   me.stations[22].raw[43,4] := WSTRING#'';
   me.stations[22].raw[43,5] := WSTRING#'';
   me.stations[22].raw[43,6] := WSTRING#'';
   me.stations[22].raw[43,7] := WSTRING#'';
   me.stations[22].raw[44,0] := WSTRING#'';
   me.stations[22].raw[44,1] := WSTRING#'';
   me.stations[22].raw[44,2] := WSTRING#'';
   me.stations[22].raw[44,3] := WSTRING#'';
   me.stations[22].raw[44,4] := WSTRING#'';
   me.stations[22].raw[44,5] := WSTRING#'';
   me.stations[22].raw[44,6] := WSTRING#'';
   me.stations[22].raw[44,7] := WSTRING#'';
   me.stations[22].raw[45,0] := WSTRING#'';
   me.stations[22].raw[45,1] := WSTRING#'';
   me.stations[22].raw[45,2] := WSTRING#'';
   me.stations[22].raw[45,3] := WSTRING#'';
   me.stations[22].raw[45,4] := WSTRING#'';
   me.stations[22].raw[45,5] := WSTRING#'';
   me.stations[22].raw[45,6] := WSTRING#'';
   me.stations[22].raw[45,7] := WSTRING#'';
   me.stations[22].raw[46,0] := WSTRING#'';
   me.stations[22].raw[46,1] := WSTRING#'';
   me.stations[22].raw[46,2] := WSTRING#'';
   me.stations[22].raw[46,3] := WSTRING#'';
   me.stations[22].raw[46,4] := WSTRING#'';
   me.stations[22].raw[46,5] := WSTRING#'';
   me.stations[22].raw[46,6] := WSTRING#'';
   me.stations[22].raw[46,7] := WSTRING#'';
   me.stations[22].raw[47,0] := WSTRING#'';
   me.stations[22].raw[47,1] := WSTRING#'';
   me.stations[22].raw[47,2] := WSTRING#'';
   me.stations[22].raw[47,3] := WSTRING#'';
   me.stations[22].raw[47,4] := WSTRING#'';
   me.stations[22].raw[47,5] := WSTRING#'';
   me.stations[22].raw[47,6] := WSTRING#'';
   me.stations[22].raw[47,7] := WSTRING#'';
   me.stations[22].raw[48,0] := WSTRING#'';
   me.stations[22].raw[48,1] := WSTRING#'';
   me.stations[22].raw[48,2] := WSTRING#'';
   me.stations[22].raw[48,3] := WSTRING#'';
   me.stations[22].raw[48,4] := WSTRING#'';
   me.stations[22].raw[48,5] := WSTRING#'';
   me.stations[22].raw[48,6] := WSTRING#'';
   me.stations[22].raw[48,7] := WSTRING#'';
   me.stations[22].raw[49,0] := WSTRING#'';
   me.stations[22].raw[49,1] := WSTRING#'';
   me.stations[22].raw[49,2] := WSTRING#'';
   me.stations[22].raw[49,3] := WSTRING#'';
   me.stations[22].raw[49,4] := WSTRING#'';
   me.stations[22].raw[49,5] := WSTRING#'';
   me.stations[22].raw[49,6] := WSTRING#'';
   me.stations[22].raw[49,7] := WSTRING#'';
   me.stations[23].size := 0;
   me.stations[23].wip[0] := WSTRING#'';
   me.stations[23].wip[1] := WSTRING#'';
   me.stations[23].wip[2] := WSTRING#'';
   me.stations[23].wip[3] := WSTRING#'';
   me.stations[23].wip[4] := WSTRING#'';
   me.stations[23].wip[5] := WSTRING#'';
   me.stations[23].wip[6] := WSTRING#'';
   me.stations[23].wip[7] := WSTRING#'';
   me.stations[23].wip[8] := WSTRING#'';
   me.stations[23].wip[9] := WSTRING#'';
   me.stations[23].wip[10] := WSTRING#'';
   me.stations[23].wip[11] := WSTRING#'';
   me.stations[23].wip[12] := WSTRING#'';
   me.stations[23].wip[13] := WSTRING#'';
   me.stations[23].wip[14] := WSTRING#'';
   me.stations[23].wip[15] := WSTRING#'';
   me.stations[23].wip[16] := WSTRING#'';
   me.stations[23].wip[17] := WSTRING#'';
   me.stations[23].wip[18] := WSTRING#'';
   me.stations[23].wip[19] := WSTRING#'';
   me.stations[23].wip[20] := WSTRING#'';
   me.stations[23].wip[21] := WSTRING#'';
   me.stations[23].wip[22] := WSTRING#'';
   me.stations[23].wip[23] := WSTRING#'';
   me.stations[23].wip[24] := WSTRING#'';
   me.stations[23].wip[25] := WSTRING#'';
   me.stations[23].wip[26] := WSTRING#'';
   me.stations[23].wip[27] := WSTRING#'';
   me.stations[23].wip[28] := WSTRING#'';
   me.stations[23].wip[29] := WSTRING#'';
   me.stations[23].wip[30] := WSTRING#'';
   me.stations[23].wip[31] := WSTRING#'';
   me.stations[23].wip[32] := WSTRING#'';
   me.stations[23].wip[33] := WSTRING#'';
   me.stations[23].wip[34] := WSTRING#'';
   me.stations[23].wip[35] := WSTRING#'';
   me.stations[23].wip[36] := WSTRING#'';
   me.stations[23].wip[37] := WSTRING#'';
   me.stations[23].wip[38] := WSTRING#'';
   me.stations[23].wip[39] := WSTRING#'';
   me.stations[23].wip[40] := WSTRING#'';
   me.stations[23].wip[41] := WSTRING#'';
   me.stations[23].wip[42] := WSTRING#'';
   me.stations[23].wip[43] := WSTRING#'';
   me.stations[23].wip[44] := WSTRING#'';
   me.stations[23].wip[45] := WSTRING#'';
   me.stations[23].wip[46] := WSTRING#'';
   me.stations[23].wip[47] := WSTRING#'';
   me.stations[23].wip[48] := WSTRING#'';
   me.stations[23].wip[49] := WSTRING#'';
   me.stations[23].raw[0,0] := WSTRING#'';
   me.stations[23].raw[0,1] := WSTRING#'';
   me.stations[23].raw[0,2] := WSTRING#'';
   me.stations[23].raw[0,3] := WSTRING#'';
   me.stations[23].raw[0,4] := WSTRING#'';
   me.stations[23].raw[0,5] := WSTRING#'';
   me.stations[23].raw[0,6] := WSTRING#'';
   me.stations[23].raw[0,7] := WSTRING#'';
   me.stations[23].raw[1,0] := WSTRING#'';
   me.stations[23].raw[1,1] := WSTRING#'';
   me.stations[23].raw[1,2] := WSTRING#'';
   me.stations[23].raw[1,3] := WSTRING#'';
   me.stations[23].raw[1,4] := WSTRING#'';
   me.stations[23].raw[1,5] := WSTRING#'';
   me.stations[23].raw[1,6] := WSTRING#'';
   me.stations[23].raw[1,7] := WSTRING#'';
   me.stations[23].raw[2,0] := WSTRING#'';
   me.stations[23].raw[2,1] := WSTRING#'';
   me.stations[23].raw[2,2] := WSTRING#'';
   me.stations[23].raw[2,3] := WSTRING#'';
   me.stations[23].raw[2,4] := WSTRING#'';
   me.stations[23].raw[2,5] := WSTRING#'';
   me.stations[23].raw[2,6] := WSTRING#'';
   me.stations[23].raw[2,7] := WSTRING#'';
   me.stations[23].raw[3,0] := WSTRING#'';
   me.stations[23].raw[3,1] := WSTRING#'';
   me.stations[23].raw[3,2] := WSTRING#'';
   me.stations[23].raw[3,3] := WSTRING#'';
   me.stations[23].raw[3,4] := WSTRING#'';
   me.stations[23].raw[3,5] := WSTRING#'';
   me.stations[23].raw[3,6] := WSTRING#'';
   me.stations[23].raw[3,7] := WSTRING#'';
   me.stations[23].raw[4,0] := WSTRING#'';
   me.stations[23].raw[4,1] := WSTRING#'';
   me.stations[23].raw[4,2] := WSTRING#'';
   me.stations[23].raw[4,3] := WSTRING#'';
   me.stations[23].raw[4,4] := WSTRING#'';
   me.stations[23].raw[4,5] := WSTRING#'';
   me.stations[23].raw[4,6] := WSTRING#'';
   me.stations[23].raw[4,7] := WSTRING#'';
   me.stations[23].raw[5,0] := WSTRING#'';
   me.stations[23].raw[5,1] := WSTRING#'';
   me.stations[23].raw[5,2] := WSTRING#'';
   me.stations[23].raw[5,3] := WSTRING#'';
   me.stations[23].raw[5,4] := WSTRING#'';
   me.stations[23].raw[5,5] := WSTRING#'';
   me.stations[23].raw[5,6] := WSTRING#'';
   me.stations[23].raw[5,7] := WSTRING#'';
   me.stations[23].raw[6,0] := WSTRING#'';
   me.stations[23].raw[6,1] := WSTRING#'';
   me.stations[23].raw[6,2] := WSTRING#'';
   me.stations[23].raw[6,3] := WSTRING#'';
   me.stations[23].raw[6,4] := WSTRING#'';
   me.stations[23].raw[6,5] := WSTRING#'';
   me.stations[23].raw[6,6] := WSTRING#'';
   me.stations[23].raw[6,7] := WSTRING#'';
   me.stations[23].raw[7,0] := WSTRING#'';
   me.stations[23].raw[7,1] := WSTRING#'';
   me.stations[23].raw[7,2] := WSTRING#'';
   me.stations[23].raw[7,3] := WSTRING#'';
   me.stations[23].raw[7,4] := WSTRING#'';
   me.stations[23].raw[7,5] := WSTRING#'';
   me.stations[23].raw[7,6] := WSTRING#'';
   me.stations[23].raw[7,7] := WSTRING#'';
   me.stations[23].raw[8,0] := WSTRING#'';
   me.stations[23].raw[8,1] := WSTRING#'';
   me.stations[23].raw[8,2] := WSTRING#'';
   me.stations[23].raw[8,3] := WSTRING#'';
   me.stations[23].raw[8,4] := WSTRING#'';
   me.stations[23].raw[8,5] := WSTRING#'';
   me.stations[23].raw[8,6] := WSTRING#'';
   me.stations[23].raw[8,7] := WSTRING#'';
   me.stations[23].raw[9,0] := WSTRING#'';
   me.stations[23].raw[9,1] := WSTRING#'';
   me.stations[23].raw[9,2] := WSTRING#'';
   me.stations[23].raw[9,3] := WSTRING#'';
   me.stations[23].raw[9,4] := WSTRING#'';
   me.stations[23].raw[9,5] := WSTRING#'';
   me.stations[23].raw[9,6] := WSTRING#'';
   me.stations[23].raw[9,7] := WSTRING#'';
   me.stations[23].raw[10,0] := WSTRING#'';
   me.stations[23].raw[10,1] := WSTRING#'';
   me.stations[23].raw[10,2] := WSTRING#'';
   me.stations[23].raw[10,3] := WSTRING#'';
   me.stations[23].raw[10,4] := WSTRING#'';
   me.stations[23].raw[10,5] := WSTRING#'';
   me.stations[23].raw[10,6] := WSTRING#'';
   me.stations[23].raw[10,7] := WSTRING#'';
   me.stations[23].raw[11,0] := WSTRING#'';
   me.stations[23].raw[11,1] := WSTRING#'';
   me.stations[23].raw[11,2] := WSTRING#'';
   me.stations[23].raw[11,3] := WSTRING#'';
   me.stations[23].raw[11,4] := WSTRING#'';
   me.stations[23].raw[11,5] := WSTRING#'';
   me.stations[23].raw[11,6] := WSTRING#'';
   me.stations[23].raw[11,7] := WSTRING#'';
   me.stations[23].raw[12,0] := WSTRING#'';
   me.stations[23].raw[12,1] := WSTRING#'';
   me.stations[23].raw[12,2] := WSTRING#'';
   me.stations[23].raw[12,3] := WSTRING#'';
   me.stations[23].raw[12,4] := WSTRING#'';
   me.stations[23].raw[12,5] := WSTRING#'';
   me.stations[23].raw[12,6] := WSTRING#'';
   me.stations[23].raw[12,7] := WSTRING#'';
   me.stations[23].raw[13,0] := WSTRING#'';
   me.stations[23].raw[13,1] := WSTRING#'';
   me.stations[23].raw[13,2] := WSTRING#'';
   me.stations[23].raw[13,3] := WSTRING#'';
   me.stations[23].raw[13,4] := WSTRING#'';
   me.stations[23].raw[13,5] := WSTRING#'';
   me.stations[23].raw[13,6] := WSTRING#'';
   me.stations[23].raw[13,7] := WSTRING#'';
   me.stations[23].raw[14,0] := WSTRING#'';
   me.stations[23].raw[14,1] := WSTRING#'';
   me.stations[23].raw[14,2] := WSTRING#'';
   me.stations[23].raw[14,3] := WSTRING#'';
   me.stations[23].raw[14,4] := WSTRING#'';
   me.stations[23].raw[14,5] := WSTRING#'';
   me.stations[23].raw[14,6] := WSTRING#'';
   me.stations[23].raw[14,7] := WSTRING#'';
   me.stations[23].raw[15,0] := WSTRING#'';
   me.stations[23].raw[15,1] := WSTRING#'';
   me.stations[23].raw[15,2] := WSTRING#'';
   me.stations[23].raw[15,3] := WSTRING#'';
   me.stations[23].raw[15,4] := WSTRING#'';
   me.stations[23].raw[15,5] := WSTRING#'';
   me.stations[23].raw[15,6] := WSTRING#'';
   me.stations[23].raw[15,7] := WSTRING#'';
   me.stations[23].raw[16,0] := WSTRING#'';
   me.stations[23].raw[16,1] := WSTRING#'';
   me.stations[23].raw[16,2] := WSTRING#'';
   me.stations[23].raw[16,3] := WSTRING#'';
   me.stations[23].raw[16,4] := WSTRING#'';
   me.stations[23].raw[16,5] := WSTRING#'';
   me.stations[23].raw[16,6] := WSTRING#'';
   me.stations[23].raw[16,7] := WSTRING#'';
   me.stations[23].raw[17,0] := WSTRING#'';
   me.stations[23].raw[17,1] := WSTRING#'';
   me.stations[23].raw[17,2] := WSTRING#'';
   me.stations[23].raw[17,3] := WSTRING#'';
   me.stations[23].raw[17,4] := WSTRING#'';
   me.stations[23].raw[17,5] := WSTRING#'';
   me.stations[23].raw[17,6] := WSTRING#'';
   me.stations[23].raw[17,7] := WSTRING#'';
   me.stations[23].raw[18,0] := WSTRING#'';
   me.stations[23].raw[18,1] := WSTRING#'';
   me.stations[23].raw[18,2] := WSTRING#'';
   me.stations[23].raw[18,3] := WSTRING#'';
   me.stations[23].raw[18,4] := WSTRING#'';
   me.stations[23].raw[18,5] := WSTRING#'';
   me.stations[23].raw[18,6] := WSTRING#'';
   me.stations[23].raw[18,7] := WSTRING#'';
   me.stations[23].raw[19,0] := WSTRING#'';
   me.stations[23].raw[19,1] := WSTRING#'';
   me.stations[23].raw[19,2] := WSTRING#'';
   me.stations[23].raw[19,3] := WSTRING#'';
   me.stations[23].raw[19,4] := WSTRING#'';
   me.stations[23].raw[19,5] := WSTRING#'';
   me.stations[23].raw[19,6] := WSTRING#'';
   me.stations[23].raw[19,7] := WSTRING#'';
   me.stations[23].raw[20,0] := WSTRING#'';
   me.stations[23].raw[20,1] := WSTRING#'';
   me.stations[23].raw[20,2] := WSTRING#'';
   me.stations[23].raw[20,3] := WSTRING#'';
   me.stations[23].raw[20,4] := WSTRING#'';
   me.stations[23].raw[20,5] := WSTRING#'';
   me.stations[23].raw[20,6] := WSTRING#'';
   me.stations[23].raw[20,7] := WSTRING#'';
   me.stations[23].raw[21,0] := WSTRING#'';
   me.stations[23].raw[21,1] := WSTRING#'';
   me.stations[23].raw[21,2] := WSTRING#'';
   me.stations[23].raw[21,3] := WSTRING#'';
   me.stations[23].raw[21,4] := WSTRING#'';
   me.stations[23].raw[21,5] := WSTRING#'';
   me.stations[23].raw[21,6] := WSTRING#'';
   me.stations[23].raw[21,7] := WSTRING#'';
   me.stations[23].raw[22,0] := WSTRING#'';
   me.stations[23].raw[22,1] := WSTRING#'';
   me.stations[23].raw[22,2] := WSTRING#'';
   me.stations[23].raw[22,3] := WSTRING#'';
   me.stations[23].raw[22,4] := WSTRING#'';
   me.stations[23].raw[22,5] := WSTRING#'';
   me.stations[23].raw[22,6] := WSTRING#'';
   me.stations[23].raw[22,7] := WSTRING#'';
   me.stations[23].raw[23,0] := WSTRING#'';
   me.stations[23].raw[23,1] := WSTRING#'';
   me.stations[23].raw[23,2] := WSTRING#'';
   me.stations[23].raw[23,3] := WSTRING#'';
   me.stations[23].raw[23,4] := WSTRING#'';
   me.stations[23].raw[23,5] := WSTRING#'';
   me.stations[23].raw[23,6] := WSTRING#'';
   me.stations[23].raw[23,7] := WSTRING#'';
   me.stations[23].raw[24,0] := WSTRING#'';
   me.stations[23].raw[24,1] := WSTRING#'';
   me.stations[23].raw[24,2] := WSTRING#'';
   me.stations[23].raw[24,3] := WSTRING#'';
   me.stations[23].raw[24,4] := WSTRING#'';
   me.stations[23].raw[24,5] := WSTRING#'';
   me.stations[23].raw[24,6] := WSTRING#'';
   me.stations[23].raw[24,7] := WSTRING#'';
   me.stations[23].raw[25,0] := WSTRING#'';
   me.stations[23].raw[25,1] := WSTRING#'';
   me.stations[23].raw[25,2] := WSTRING#'';
   me.stations[23].raw[25,3] := WSTRING#'';
   me.stations[23].raw[25,4] := WSTRING#'';
   me.stations[23].raw[25,5] := WSTRING#'';
   me.stations[23].raw[25,6] := WSTRING#'';
   me.stations[23].raw[25,7] := WSTRING#'';
   me.stations[23].raw[26,0] := WSTRING#'';
   me.stations[23].raw[26,1] := WSTRING#'';
   me.stations[23].raw[26,2] := WSTRING#'';
   me.stations[23].raw[26,3] := WSTRING#'';
   me.stations[23].raw[26,4] := WSTRING#'';
   me.stations[23].raw[26,5] := WSTRING#'';
   me.stations[23].raw[26,6] := WSTRING#'';
   me.stations[23].raw[26,7] := WSTRING#'';
   me.stations[23].raw[27,0] := WSTRING#'';
   me.stations[23].raw[27,1] := WSTRING#'';
   me.stations[23].raw[27,2] := WSTRING#'';
   me.stations[23].raw[27,3] := WSTRING#'';
   me.stations[23].raw[27,4] := WSTRING#'';
   me.stations[23].raw[27,5] := WSTRING#'';
   me.stations[23].raw[27,6] := WSTRING#'';
   me.stations[23].raw[27,7] := WSTRING#'';
   me.stations[23].raw[28,0] := WSTRING#'';
   me.stations[23].raw[28,1] := WSTRING#'';
   me.stations[23].raw[28,2] := WSTRING#'';
   me.stations[23].raw[28,3] := WSTRING#'';
   me.stations[23].raw[28,4] := WSTRING#'';
   me.stations[23].raw[28,5] := WSTRING#'';
   me.stations[23].raw[28,6] := WSTRING#'';
   me.stations[23].raw[28,7] := WSTRING#'';
   me.stations[23].raw[29,0] := WSTRING#'';
   me.stations[23].raw[29,1] := WSTRING#'';
   me.stations[23].raw[29,2] := WSTRING#'';
   me.stations[23].raw[29,3] := WSTRING#'';
   me.stations[23].raw[29,4] := WSTRING#'';
   me.stations[23].raw[29,5] := WSTRING#'';
   me.stations[23].raw[29,6] := WSTRING#'';
   me.stations[23].raw[29,7] := WSTRING#'';
   me.stations[23].raw[30,0] := WSTRING#'';
   me.stations[23].raw[30,1] := WSTRING#'';
   me.stations[23].raw[30,2] := WSTRING#'';
   me.stations[23].raw[30,3] := WSTRING#'';
   me.stations[23].raw[30,4] := WSTRING#'';
   me.stations[23].raw[30,5] := WSTRING#'';
   me.stations[23].raw[30,6] := WSTRING#'';
   me.stations[23].raw[30,7] := WSTRING#'';
   me.stations[23].raw[31,0] := WSTRING#'';
   me.stations[23].raw[31,1] := WSTRING#'';
   me.stations[23].raw[31,2] := WSTRING#'';
   me.stations[23].raw[31,3] := WSTRING#'';
   me.stations[23].raw[31,4] := WSTRING#'';
   me.stations[23].raw[31,5] := WSTRING#'';
   me.stations[23].raw[31,6] := WSTRING#'';
   me.stations[23].raw[31,7] := WSTRING#'';
   me.stations[23].raw[32,0] := WSTRING#'';
   me.stations[23].raw[32,1] := WSTRING#'';
   me.stations[23].raw[32,2] := WSTRING#'';
   me.stations[23].raw[32,3] := WSTRING#'';
   me.stations[23].raw[32,4] := WSTRING#'';
   me.stations[23].raw[32,5] := WSTRING#'';
   me.stations[23].raw[32,6] := WSTRING#'';
   me.stations[23].raw[32,7] := WSTRING#'';
   me.stations[23].raw[33,0] := WSTRING#'';
   me.stations[23].raw[33,1] := WSTRING#'';
   me.stations[23].raw[33,2] := WSTRING#'';
   me.stations[23].raw[33,3] := WSTRING#'';
   me.stations[23].raw[33,4] := WSTRING#'';
   me.stations[23].raw[33,5] := WSTRING#'';
   me.stations[23].raw[33,6] := WSTRING#'';
   me.stations[23].raw[33,7] := WSTRING#'';
   me.stations[23].raw[34,0] := WSTRING#'';
   me.stations[23].raw[34,1] := WSTRING#'';
   me.stations[23].raw[34,2] := WSTRING#'';
   me.stations[23].raw[34,3] := WSTRING#'';
   me.stations[23].raw[34,4] := WSTRING#'';
   me.stations[23].raw[34,5] := WSTRING#'';
   me.stations[23].raw[34,6] := WSTRING#'';
   me.stations[23].raw[34,7] := WSTRING#'';
   me.stations[23].raw[35,0] := WSTRING#'';
   me.stations[23].raw[35,1] := WSTRING#'';
   me.stations[23].raw[35,2] := WSTRING#'';
   me.stations[23].raw[35,3] := WSTRING#'';
   me.stations[23].raw[35,4] := WSTRING#'';
   me.stations[23].raw[35,5] := WSTRING#'';
   me.stations[23].raw[35,6] := WSTRING#'';
   me.stations[23].raw[35,7] := WSTRING#'';
   me.stations[23].raw[36,0] := WSTRING#'';
   me.stations[23].raw[36,1] := WSTRING#'';
   me.stations[23].raw[36,2] := WSTRING#'';
   me.stations[23].raw[36,3] := WSTRING#'';
   me.stations[23].raw[36,4] := WSTRING#'';
   me.stations[23].raw[36,5] := WSTRING#'';
   me.stations[23].raw[36,6] := WSTRING#'';
   me.stations[23].raw[36,7] := WSTRING#'';
   me.stations[23].raw[37,0] := WSTRING#'';
   me.stations[23].raw[37,1] := WSTRING#'';
   me.stations[23].raw[37,2] := WSTRING#'';
   me.stations[23].raw[37,3] := WSTRING#'';
   me.stations[23].raw[37,4] := WSTRING#'';
   me.stations[23].raw[37,5] := WSTRING#'';
   me.stations[23].raw[37,6] := WSTRING#'';
   me.stations[23].raw[37,7] := WSTRING#'';
   me.stations[23].raw[38,0] := WSTRING#'';
   me.stations[23].raw[38,1] := WSTRING#'';
   me.stations[23].raw[38,2] := WSTRING#'';
   me.stations[23].raw[38,3] := WSTRING#'';
   me.stations[23].raw[38,4] := WSTRING#'';
   me.stations[23].raw[38,5] := WSTRING#'';
   me.stations[23].raw[38,6] := WSTRING#'';
   me.stations[23].raw[38,7] := WSTRING#'';
   me.stations[23].raw[39,0] := WSTRING#'';
   me.stations[23].raw[39,1] := WSTRING#'';
   me.stations[23].raw[39,2] := WSTRING#'';
   me.stations[23].raw[39,3] := WSTRING#'';
   me.stations[23].raw[39,4] := WSTRING#'';
   me.stations[23].raw[39,5] := WSTRING#'';
   me.stations[23].raw[39,6] := WSTRING#'';
   me.stations[23].raw[39,7] := WSTRING#'';
   me.stations[23].raw[40,0] := WSTRING#'';
   me.stations[23].raw[40,1] := WSTRING#'';
   me.stations[23].raw[40,2] := WSTRING#'';
   me.stations[23].raw[40,3] := WSTRING#'';
   me.stations[23].raw[40,4] := WSTRING#'';
   me.stations[23].raw[40,5] := WSTRING#'';
   me.stations[23].raw[40,6] := WSTRING#'';
   me.stations[23].raw[40,7] := WSTRING#'';
   me.stations[23].raw[41,0] := WSTRING#'';
   me.stations[23].raw[41,1] := WSTRING#'';
   me.stations[23].raw[41,2] := WSTRING#'';
   me.stations[23].raw[41,3] := WSTRING#'';
   me.stations[23].raw[41,4] := WSTRING#'';
   me.stations[23].raw[41,5] := WSTRING#'';
   me.stations[23].raw[41,6] := WSTRING#'';
   me.stations[23].raw[41,7] := WSTRING#'';
   me.stations[23].raw[42,0] := WSTRING#'';
   me.stations[23].raw[42,1] := WSTRING#'';
   me.stations[23].raw[42,2] := WSTRING#'';
   me.stations[23].raw[42,3] := WSTRING#'';
   me.stations[23].raw[42,4] := WSTRING#'';
   me.stations[23].raw[42,5] := WSTRING#'';
   me.stations[23].raw[42,6] := WSTRING#'';
   me.stations[23].raw[42,7] := WSTRING#'';
   me.stations[23].raw[43,0] := WSTRING#'';
   me.stations[23].raw[43,1] := WSTRING#'';
   me.stations[23].raw[43,2] := WSTRING#'';
   me.stations[23].raw[43,3] := WSTRING#'';
   me.stations[23].raw[43,4] := WSTRING#'';
   me.stations[23].raw[43,5] := WSTRING#'';
   me.stations[23].raw[43,6] := WSTRING#'';
   me.stations[23].raw[43,7] := WSTRING#'';
   me.stations[23].raw[44,0] := WSTRING#'';
   me.stations[23].raw[44,1] := WSTRING#'';
   me.stations[23].raw[44,2] := WSTRING#'';
   me.stations[23].raw[44,3] := WSTRING#'';
   me.stations[23].raw[44,4] := WSTRING#'';
   me.stations[23].raw[44,5] := WSTRING#'';
   me.stations[23].raw[44,6] := WSTRING#'';
   me.stations[23].raw[44,7] := WSTRING#'';
   me.stations[23].raw[45,0] := WSTRING#'';
   me.stations[23].raw[45,1] := WSTRING#'';
   me.stations[23].raw[45,2] := WSTRING#'';
   me.stations[23].raw[45,3] := WSTRING#'';
   me.stations[23].raw[45,4] := WSTRING#'';
   me.stations[23].raw[45,5] := WSTRING#'';
   me.stations[23].raw[45,6] := WSTRING#'';
   me.stations[23].raw[45,7] := WSTRING#'';
   me.stations[23].raw[46,0] := WSTRING#'';
   me.stations[23].raw[46,1] := WSTRING#'';
   me.stations[23].raw[46,2] := WSTRING#'';
   me.stations[23].raw[46,3] := WSTRING#'';
   me.stations[23].raw[46,4] := WSTRING#'';
   me.stations[23].raw[46,5] := WSTRING#'';
   me.stations[23].raw[46,6] := WSTRING#'';
   me.stations[23].raw[46,7] := WSTRING#'';
   me.stations[23].raw[47,0] := WSTRING#'';
   me.stations[23].raw[47,1] := WSTRING#'';
   me.stations[23].raw[47,2] := WSTRING#'';
   me.stations[23].raw[47,3] := WSTRING#'';
   me.stations[23].raw[47,4] := WSTRING#'';
   me.stations[23].raw[47,5] := WSTRING#'';
   me.stations[23].raw[47,6] := WSTRING#'';
   me.stations[23].raw[47,7] := WSTRING#'';
   me.stations[23].raw[48,0] := WSTRING#'';
   me.stations[23].raw[48,1] := WSTRING#'';
   me.stations[23].raw[48,2] := WSTRING#'';
   me.stations[23].raw[48,3] := WSTRING#'';
   me.stations[23].raw[48,4] := WSTRING#'';
   me.stations[23].raw[48,5] := WSTRING#'';
   me.stations[23].raw[48,6] := WSTRING#'';
   me.stations[23].raw[48,7] := WSTRING#'';
   me.stations[23].raw[49,0] := WSTRING#'';
   me.stations[23].raw[49,1] := WSTRING#'';
   me.stations[23].raw[49,2] := WSTRING#'';
   me.stations[23].raw[49,3] := WSTRING#'';
   me.stations[23].raw[49,4] := WSTRING#'';
   me.stations[23].raw[49,5] := WSTRING#'';
   me.stations[23].raw[49,6] := WSTRING#'';
   me.stations[23].raw[49,7] := WSTRING#'';
   me.stations[24].size := 0;
   me.stations[24].wip[0] := WSTRING#'';
   me.stations[24].wip[1] := WSTRING#'';
   me.stations[24].wip[2] := WSTRING#'';
   me.stations[24].wip[3] := WSTRING#'';
   me.stations[24].wip[4] := WSTRING#'';
   me.stations[24].wip[5] := WSTRING#'';
   me.stations[24].wip[6] := WSTRING#'';
   me.stations[24].wip[7] := WSTRING#'';
   me.stations[24].wip[8] := WSTRING#'';
   me.stations[24].wip[9] := WSTRING#'';
   me.stations[24].wip[10] := WSTRING#'';
   me.stations[24].wip[11] := WSTRING#'';
   me.stations[24].wip[12] := WSTRING#'';
   me.stations[24].wip[13] := WSTRING#'';
   me.stations[24].wip[14] := WSTRING#'';
   me.stations[24].wip[15] := WSTRING#'';
   me.stations[24].wip[16] := WSTRING#'';
   me.stations[24].wip[17] := WSTRING#'';
   me.stations[24].wip[18] := WSTRING#'';
   me.stations[24].wip[19] := WSTRING#'';
   me.stations[24].wip[20] := WSTRING#'';
   me.stations[24].wip[21] := WSTRING#'';
   me.stations[24].wip[22] := WSTRING#'';
   me.stations[24].wip[23] := WSTRING#'';
   me.stations[24].wip[24] := WSTRING#'';
   me.stations[24].wip[25] := WSTRING#'';
   me.stations[24].wip[26] := WSTRING#'';
   me.stations[24].wip[27] := WSTRING#'';
   me.stations[24].wip[28] := WSTRING#'';
   me.stations[24].wip[29] := WSTRING#'';
   me.stations[24].wip[30] := WSTRING#'';
   me.stations[24].wip[31] := WSTRING#'';
   me.stations[24].wip[32] := WSTRING#'';
   me.stations[24].wip[33] := WSTRING#'';
   me.stations[24].wip[34] := WSTRING#'';
   me.stations[24].wip[35] := WSTRING#'';
   me.stations[24].wip[36] := WSTRING#'';
   me.stations[24].wip[37] := WSTRING#'';
   me.stations[24].wip[38] := WSTRING#'';
   me.stations[24].wip[39] := WSTRING#'';
   me.stations[24].wip[40] := WSTRING#'';
   me.stations[24].wip[41] := WSTRING#'';
   me.stations[24].wip[42] := WSTRING#'';
   me.stations[24].wip[43] := WSTRING#'';
   me.stations[24].wip[44] := WSTRING#'';
   me.stations[24].wip[45] := WSTRING#'';
   me.stations[24].wip[46] := WSTRING#'';
   me.stations[24].wip[47] := WSTRING#'';
   me.stations[24].wip[48] := WSTRING#'';
   me.stations[24].wip[49] := WSTRING#'';
   me.stations[24].raw[0,0] := WSTRING#'';
   me.stations[24].raw[0,1] := WSTRING#'';
   me.stations[24].raw[0,2] := WSTRING#'';
   me.stations[24].raw[0,3] := WSTRING#'';
   me.stations[24].raw[0,4] := WSTRING#'';
   me.stations[24].raw[0,5] := WSTRING#'';
   me.stations[24].raw[0,6] := WSTRING#'';
   me.stations[24].raw[0,7] := WSTRING#'';
   me.stations[24].raw[1,0] := WSTRING#'';
   me.stations[24].raw[1,1] := WSTRING#'';
   me.stations[24].raw[1,2] := WSTRING#'';
   me.stations[24].raw[1,3] := WSTRING#'';
   me.stations[24].raw[1,4] := WSTRING#'';
   me.stations[24].raw[1,5] := WSTRING#'';
   me.stations[24].raw[1,6] := WSTRING#'';
   me.stations[24].raw[1,7] := WSTRING#'';
   me.stations[24].raw[2,0] := WSTRING#'';
   me.stations[24].raw[2,1] := WSTRING#'';
   me.stations[24].raw[2,2] := WSTRING#'';
   me.stations[24].raw[2,3] := WSTRING#'';
   me.stations[24].raw[2,4] := WSTRING#'';
   me.stations[24].raw[2,5] := WSTRING#'';
   me.stations[24].raw[2,6] := WSTRING#'';
   me.stations[24].raw[2,7] := WSTRING#'';
   me.stations[24].raw[3,0] := WSTRING#'';
   me.stations[24].raw[3,1] := WSTRING#'';
   me.stations[24].raw[3,2] := WSTRING#'';
   me.stations[24].raw[3,3] := WSTRING#'';
   me.stations[24].raw[3,4] := WSTRING#'';
   me.stations[24].raw[3,5] := WSTRING#'';
   me.stations[24].raw[3,6] := WSTRING#'';
   me.stations[24].raw[3,7] := WSTRING#'';
   me.stations[24].raw[4,0] := WSTRING#'';
   me.stations[24].raw[4,1] := WSTRING#'';
   me.stations[24].raw[4,2] := WSTRING#'';
   me.stations[24].raw[4,3] := WSTRING#'';
   me.stations[24].raw[4,4] := WSTRING#'';
   me.stations[24].raw[4,5] := WSTRING#'';
   me.stations[24].raw[4,6] := WSTRING#'';
   me.stations[24].raw[4,7] := WSTRING#'';
   me.stations[24].raw[5,0] := WSTRING#'';
   me.stations[24].raw[5,1] := WSTRING#'';
   me.stations[24].raw[5,2] := WSTRING#'';
   me.stations[24].raw[5,3] := WSTRING#'';
   me.stations[24].raw[5,4] := WSTRING#'';
   me.stations[24].raw[5,5] := WSTRING#'';
   me.stations[24].raw[5,6] := WSTRING#'';
   me.stations[24].raw[5,7] := WSTRING#'';
   me.stations[24].raw[6,0] := WSTRING#'';
   me.stations[24].raw[6,1] := WSTRING#'';
   me.stations[24].raw[6,2] := WSTRING#'';
   me.stations[24].raw[6,3] := WSTRING#'';
   me.stations[24].raw[6,4] := WSTRING#'';
   me.stations[24].raw[6,5] := WSTRING#'';
   me.stations[24].raw[6,6] := WSTRING#'';
   me.stations[24].raw[6,7] := WSTRING#'';
   me.stations[24].raw[7,0] := WSTRING#'';
   me.stations[24].raw[7,1] := WSTRING#'';
   me.stations[24].raw[7,2] := WSTRING#'';
   me.stations[24].raw[7,3] := WSTRING#'';
   me.stations[24].raw[7,4] := WSTRING#'';
   me.stations[24].raw[7,5] := WSTRING#'';
   me.stations[24].raw[7,6] := WSTRING#'';
   me.stations[24].raw[7,7] := WSTRING#'';
   me.stations[24].raw[8,0] := WSTRING#'';
   me.stations[24].raw[8,1] := WSTRING#'';
   me.stations[24].raw[8,2] := WSTRING#'';
   me.stations[24].raw[8,3] := WSTRING#'';
   me.stations[24].raw[8,4] := WSTRING#'';
   me.stations[24].raw[8,5] := WSTRING#'';
   me.stations[24].raw[8,6] := WSTRING#'';
   me.stations[24].raw[8,7] := WSTRING#'';
   me.stations[24].raw[9,0] := WSTRING#'';
   me.stations[24].raw[9,1] := WSTRING#'';
   me.stations[24].raw[9,2] := WSTRING#'';
   me.stations[24].raw[9,3] := WSTRING#'';
   me.stations[24].raw[9,4] := WSTRING#'';
   me.stations[24].raw[9,5] := WSTRING#'';
   me.stations[24].raw[9,6] := WSTRING#'';
   me.stations[24].raw[9,7] := WSTRING#'';
   me.stations[24].raw[10,0] := WSTRING#'';
   me.stations[24].raw[10,1] := WSTRING#'';
   me.stations[24].raw[10,2] := WSTRING#'';
   me.stations[24].raw[10,3] := WSTRING#'';
   me.stations[24].raw[10,4] := WSTRING#'';
   me.stations[24].raw[10,5] := WSTRING#'';
   me.stations[24].raw[10,6] := WSTRING#'';
   me.stations[24].raw[10,7] := WSTRING#'';
   me.stations[24].raw[11,0] := WSTRING#'';
   me.stations[24].raw[11,1] := WSTRING#'';
   me.stations[24].raw[11,2] := WSTRING#'';
   me.stations[24].raw[11,3] := WSTRING#'';
   me.stations[24].raw[11,4] := WSTRING#'';
   me.stations[24].raw[11,5] := WSTRING#'';
   me.stations[24].raw[11,6] := WSTRING#'';
   me.stations[24].raw[11,7] := WSTRING#'';
   me.stations[24].raw[12,0] := WSTRING#'';
   me.stations[24].raw[12,1] := WSTRING#'';
   me.stations[24].raw[12,2] := WSTRING#'';
   me.stations[24].raw[12,3] := WSTRING#'';
   me.stations[24].raw[12,4] := WSTRING#'';
   me.stations[24].raw[12,5] := WSTRING#'';
   me.stations[24].raw[12,6] := WSTRING#'';
   me.stations[24].raw[12,7] := WSTRING#'';
   me.stations[24].raw[13,0] := WSTRING#'';
   me.stations[24].raw[13,1] := WSTRING#'';
   me.stations[24].raw[13,2] := WSTRING#'';
   me.stations[24].raw[13,3] := WSTRING#'';
   me.stations[24].raw[13,4] := WSTRING#'';
   me.stations[24].raw[13,5] := WSTRING#'';
   me.stations[24].raw[13,6] := WSTRING#'';
   me.stations[24].raw[13,7] := WSTRING#'';
   me.stations[24].raw[14,0] := WSTRING#'';
   me.stations[24].raw[14,1] := WSTRING#'';
   me.stations[24].raw[14,2] := WSTRING#'';
   me.stations[24].raw[14,3] := WSTRING#'';
   me.stations[24].raw[14,4] := WSTRING#'';
   me.stations[24].raw[14,5] := WSTRING#'';
   me.stations[24].raw[14,6] := WSTRING#'';
   me.stations[24].raw[14,7] := WSTRING#'';
   me.stations[24].raw[15,0] := WSTRING#'';
   me.stations[24].raw[15,1] := WSTRING#'';
   me.stations[24].raw[15,2] := WSTRING#'';
   me.stations[24].raw[15,3] := WSTRING#'';
   me.stations[24].raw[15,4] := WSTRING#'';
   me.stations[24].raw[15,5] := WSTRING#'';
   me.stations[24].raw[15,6] := WSTRING#'';
   me.stations[24].raw[15,7] := WSTRING#'';
   me.stations[24].raw[16,0] := WSTRING#'';
   me.stations[24].raw[16,1] := WSTRING#'';
   me.stations[24].raw[16,2] := WSTRING#'';
   me.stations[24].raw[16,3] := WSTRING#'';
   me.stations[24].raw[16,4] := WSTRING#'';
   me.stations[24].raw[16,5] := WSTRING#'';
   me.stations[24].raw[16,6] := WSTRING#'';
   me.stations[24].raw[16,7] := WSTRING#'';
   me.stations[24].raw[17,0] := WSTRING#'';
   me.stations[24].raw[17,1] := WSTRING#'';
   me.stations[24].raw[17,2] := WSTRING#'';
   me.stations[24].raw[17,3] := WSTRING#'';
   me.stations[24].raw[17,4] := WSTRING#'';
   me.stations[24].raw[17,5] := WSTRING#'';
   me.stations[24].raw[17,6] := WSTRING#'';
   me.stations[24].raw[17,7] := WSTRING#'';
   me.stations[24].raw[18,0] := WSTRING#'';
   me.stations[24].raw[18,1] := WSTRING#'';
   me.stations[24].raw[18,2] := WSTRING#'';
   me.stations[24].raw[18,3] := WSTRING#'';
   me.stations[24].raw[18,4] := WSTRING#'';
   me.stations[24].raw[18,5] := WSTRING#'';
   me.stations[24].raw[18,6] := WSTRING#'';
   me.stations[24].raw[18,7] := WSTRING#'';
   me.stations[24].raw[19,0] := WSTRING#'';
   me.stations[24].raw[19,1] := WSTRING#'';
   me.stations[24].raw[19,2] := WSTRING#'';
   me.stations[24].raw[19,3] := WSTRING#'';
   me.stations[24].raw[19,4] := WSTRING#'';
   me.stations[24].raw[19,5] := WSTRING#'';
   me.stations[24].raw[19,6] := WSTRING#'';
   me.stations[24].raw[19,7] := WSTRING#'';
   me.stations[24].raw[20,0] := WSTRING#'';
   me.stations[24].raw[20,1] := WSTRING#'';
   me.stations[24].raw[20,2] := WSTRING#'';
   me.stations[24].raw[20,3] := WSTRING#'';
   me.stations[24].raw[20,4] := WSTRING#'';
   me.stations[24].raw[20,5] := WSTRING#'';
   me.stations[24].raw[20,6] := WSTRING#'';
   me.stations[24].raw[20,7] := WSTRING#'';
   me.stations[24].raw[21,0] := WSTRING#'';
   me.stations[24].raw[21,1] := WSTRING#'';
   me.stations[24].raw[21,2] := WSTRING#'';
   me.stations[24].raw[21,3] := WSTRING#'';
   me.stations[24].raw[21,4] := WSTRING#'';
   me.stations[24].raw[21,5] := WSTRING#'';
   me.stations[24].raw[21,6] := WSTRING#'';
   me.stations[24].raw[21,7] := WSTRING#'';
   me.stations[24].raw[22,0] := WSTRING#'';
   me.stations[24].raw[22,1] := WSTRING#'';
   me.stations[24].raw[22,2] := WSTRING#'';
   me.stations[24].raw[22,3] := WSTRING#'';
   me.stations[24].raw[22,4] := WSTRING#'';
   me.stations[24].raw[22,5] := WSTRING#'';
   me.stations[24].raw[22,6] := WSTRING#'';
   me.stations[24].raw[22,7] := WSTRING#'';
   me.stations[24].raw[23,0] := WSTRING#'';
   me.stations[24].raw[23,1] := WSTRING#'';
   me.stations[24].raw[23,2] := WSTRING#'';
   me.stations[24].raw[23,3] := WSTRING#'';
   me.stations[24].raw[23,4] := WSTRING#'';
   me.stations[24].raw[23,5] := WSTRING#'';
   me.stations[24].raw[23,6] := WSTRING#'';
   me.stations[24].raw[23,7] := WSTRING#'';
   me.stations[24].raw[24,0] := WSTRING#'';
   me.stations[24].raw[24,1] := WSTRING#'';
   me.stations[24].raw[24,2] := WSTRING#'';
   me.stations[24].raw[24,3] := WSTRING#'';
   me.stations[24].raw[24,4] := WSTRING#'';
   me.stations[24].raw[24,5] := WSTRING#'';
   me.stations[24].raw[24,6] := WSTRING#'';
   me.stations[24].raw[24,7] := WSTRING#'';
   me.stations[24].raw[25,0] := WSTRING#'';
   me.stations[24].raw[25,1] := WSTRING#'';
   me.stations[24].raw[25,2] := WSTRING#'';
   me.stations[24].raw[25,3] := WSTRING#'';
   me.stations[24].raw[25,4] := WSTRING#'';
   me.stations[24].raw[25,5] := WSTRING#'';
   me.stations[24].raw[25,6] := WSTRING#'';
   me.stations[24].raw[25,7] := WSTRING#'';
   me.stations[24].raw[26,0] := WSTRING#'';
   me.stations[24].raw[26,1] := WSTRING#'';
   me.stations[24].raw[26,2] := WSTRING#'';
   me.stations[24].raw[26,3] := WSTRING#'';
   me.stations[24].raw[26,4] := WSTRING#'';
   me.stations[24].raw[26,5] := WSTRING#'';
   me.stations[24].raw[26,6] := WSTRING#'';
   me.stations[24].raw[26,7] := WSTRING#'';
   me.stations[24].raw[27,0] := WSTRING#'';
   me.stations[24].raw[27,1] := WSTRING#'';
   me.stations[24].raw[27,2] := WSTRING#'';
   me.stations[24].raw[27,3] := WSTRING#'';
   me.stations[24].raw[27,4] := WSTRING#'';
   me.stations[24].raw[27,5] := WSTRING#'';
   me.stations[24].raw[27,6] := WSTRING#'';
   me.stations[24].raw[27,7] := WSTRING#'';
   me.stations[24].raw[28,0] := WSTRING#'';
   me.stations[24].raw[28,1] := WSTRING#'';
   me.stations[24].raw[28,2] := WSTRING#'';
   me.stations[24].raw[28,3] := WSTRING#'';
   me.stations[24].raw[28,4] := WSTRING#'';
   me.stations[24].raw[28,5] := WSTRING#'';
   me.stations[24].raw[28,6] := WSTRING#'';
   me.stations[24].raw[28,7] := WSTRING#'';
   me.stations[24].raw[29,0] := WSTRING#'';
   me.stations[24].raw[29,1] := WSTRING#'';
   me.stations[24].raw[29,2] := WSTRING#'';
   me.stations[24].raw[29,3] := WSTRING#'';
   me.stations[24].raw[29,4] := WSTRING#'';
   me.stations[24].raw[29,5] := WSTRING#'';
   me.stations[24].raw[29,6] := WSTRING#'';
   me.stations[24].raw[29,7] := WSTRING#'';
   me.stations[24].raw[30,0] := WSTRING#'';
   me.stations[24].raw[30,1] := WSTRING#'';
   me.stations[24].raw[30,2] := WSTRING#'';
   me.stations[24].raw[30,3] := WSTRING#'';
   me.stations[24].raw[30,4] := WSTRING#'';
   me.stations[24].raw[30,5] := WSTRING#'';
   me.stations[24].raw[30,6] := WSTRING#'';
   me.stations[24].raw[30,7] := WSTRING#'';
   me.stations[24].raw[31,0] := WSTRING#'';
   me.stations[24].raw[31,1] := WSTRING#'';
   me.stations[24].raw[31,2] := WSTRING#'';
   me.stations[24].raw[31,3] := WSTRING#'';
   me.stations[24].raw[31,4] := WSTRING#'';
   me.stations[24].raw[31,5] := WSTRING#'';
   me.stations[24].raw[31,6] := WSTRING#'';
   me.stations[24].raw[31,7] := WSTRING#'';
   me.stations[24].raw[32,0] := WSTRING#'';
   me.stations[24].raw[32,1] := WSTRING#'';
   me.stations[24].raw[32,2] := WSTRING#'';
   me.stations[24].raw[32,3] := WSTRING#'';
   me.stations[24].raw[32,4] := WSTRING#'';
   me.stations[24].raw[32,5] := WSTRING#'';
   me.stations[24].raw[32,6] := WSTRING#'';
   me.stations[24].raw[32,7] := WSTRING#'';
   me.stations[24].raw[33,0] := WSTRING#'';
   me.stations[24].raw[33,1] := WSTRING#'';
   me.stations[24].raw[33,2] := WSTRING#'';
   me.stations[24].raw[33,3] := WSTRING#'';
   me.stations[24].raw[33,4] := WSTRING#'';
   me.stations[24].raw[33,5] := WSTRING#'';
   me.stations[24].raw[33,6] := WSTRING#'';
   me.stations[24].raw[33,7] := WSTRING#'';
   me.stations[24].raw[34,0] := WSTRING#'';
   me.stations[24].raw[34,1] := WSTRING#'';
   me.stations[24].raw[34,2] := WSTRING#'';
   me.stations[24].raw[34,3] := WSTRING#'';
   me.stations[24].raw[34,4] := WSTRING#'';
   me.stations[24].raw[34,5] := WSTRING#'';
   me.stations[24].raw[34,6] := WSTRING#'';
   me.stations[24].raw[34,7] := WSTRING#'';
   me.stations[24].raw[35,0] := WSTRING#'';
   me.stations[24].raw[35,1] := WSTRING#'';
   me.stations[24].raw[35,2] := WSTRING#'';
   me.stations[24].raw[35,3] := WSTRING#'';
   me.stations[24].raw[35,4] := WSTRING#'';
   me.stations[24].raw[35,5] := WSTRING#'';
   me.stations[24].raw[35,6] := WSTRING#'';
   me.stations[24].raw[35,7] := WSTRING#'';
   me.stations[24].raw[36,0] := WSTRING#'';
   me.stations[24].raw[36,1] := WSTRING#'';
   me.stations[24].raw[36,2] := WSTRING#'';
   me.stations[24].raw[36,3] := WSTRING#'';
   me.stations[24].raw[36,4] := WSTRING#'';
   me.stations[24].raw[36,5] := WSTRING#'';
   me.stations[24].raw[36,6] := WSTRING#'';
   me.stations[24].raw[36,7] := WSTRING#'';
   me.stations[24].raw[37,0] := WSTRING#'';
   me.stations[24].raw[37,1] := WSTRING#'';
   me.stations[24].raw[37,2] := WSTRING#'';
   me.stations[24].raw[37,3] := WSTRING#'';
   me.stations[24].raw[37,4] := WSTRING#'';
   me.stations[24].raw[37,5] := WSTRING#'';
   me.stations[24].raw[37,6] := WSTRING#'';
   me.stations[24].raw[37,7] := WSTRING#'';
   me.stations[24].raw[38,0] := WSTRING#'';
   me.stations[24].raw[38,1] := WSTRING#'';
   me.stations[24].raw[38,2] := WSTRING#'';
   me.stations[24].raw[38,3] := WSTRING#'';
   me.stations[24].raw[38,4] := WSTRING#'';
   me.stations[24].raw[38,5] := WSTRING#'';
   me.stations[24].raw[38,6] := WSTRING#'';
   me.stations[24].raw[38,7] := WSTRING#'';
   me.stations[24].raw[39,0] := WSTRING#'';
   me.stations[24].raw[39,1] := WSTRING#'';
   me.stations[24].raw[39,2] := WSTRING#'';
   me.stations[24].raw[39,3] := WSTRING#'';
   me.stations[24].raw[39,4] := WSTRING#'';
   me.stations[24].raw[39,5] := WSTRING#'';
   me.stations[24].raw[39,6] := WSTRING#'';
   me.stations[24].raw[39,7] := WSTRING#'';
   me.stations[24].raw[40,0] := WSTRING#'';
   me.stations[24].raw[40,1] := WSTRING#'';
   me.stations[24].raw[40,2] := WSTRING#'';
   me.stations[24].raw[40,3] := WSTRING#'';
   me.stations[24].raw[40,4] := WSTRING#'';
   me.stations[24].raw[40,5] := WSTRING#'';
   me.stations[24].raw[40,6] := WSTRING#'';
   me.stations[24].raw[40,7] := WSTRING#'';
   me.stations[24].raw[41,0] := WSTRING#'';
   me.stations[24].raw[41,1] := WSTRING#'';
   me.stations[24].raw[41,2] := WSTRING#'';
   me.stations[24].raw[41,3] := WSTRING#'';
   me.stations[24].raw[41,4] := WSTRING#'';
   me.stations[24].raw[41,5] := WSTRING#'';
   me.stations[24].raw[41,6] := WSTRING#'';
   me.stations[24].raw[41,7] := WSTRING#'';
   me.stations[24].raw[42,0] := WSTRING#'';
   me.stations[24].raw[42,1] := WSTRING#'';
   me.stations[24].raw[42,2] := WSTRING#'';
   me.stations[24].raw[42,3] := WSTRING#'';
   me.stations[24].raw[42,4] := WSTRING#'';
   me.stations[24].raw[42,5] := WSTRING#'';
   me.stations[24].raw[42,6] := WSTRING#'';
   me.stations[24].raw[42,7] := WSTRING#'';
   me.stations[24].raw[43,0] := WSTRING#'';
   me.stations[24].raw[43,1] := WSTRING#'';
   me.stations[24].raw[43,2] := WSTRING#'';
   me.stations[24].raw[43,3] := WSTRING#'';
   me.stations[24].raw[43,4] := WSTRING#'';
   me.stations[24].raw[43,5] := WSTRING#'';
   me.stations[24].raw[43,6] := WSTRING#'';
   me.stations[24].raw[43,7] := WSTRING#'';
   me.stations[24].raw[44,0] := WSTRING#'';
   me.stations[24].raw[44,1] := WSTRING#'';
   me.stations[24].raw[44,2] := WSTRING#'';
   me.stations[24].raw[44,3] := WSTRING#'';
   me.stations[24].raw[44,4] := WSTRING#'';
   me.stations[24].raw[44,5] := WSTRING#'';
   me.stations[24].raw[44,6] := WSTRING#'';
   me.stations[24].raw[44,7] := WSTRING#'';
   me.stations[24].raw[45,0] := WSTRING#'';
   me.stations[24].raw[45,1] := WSTRING#'';
   me.stations[24].raw[45,2] := WSTRING#'';
   me.stations[24].raw[45,3] := WSTRING#'';
   me.stations[24].raw[45,4] := WSTRING#'';
   me.stations[24].raw[45,5] := WSTRING#'';
   me.stations[24].raw[45,6] := WSTRING#'';
   me.stations[24].raw[45,7] := WSTRING#'';
   me.stations[24].raw[46,0] := WSTRING#'';
   me.stations[24].raw[46,1] := WSTRING#'';
   me.stations[24].raw[46,2] := WSTRING#'';
   me.stations[24].raw[46,3] := WSTRING#'';
   me.stations[24].raw[46,4] := WSTRING#'';
   me.stations[24].raw[46,5] := WSTRING#'';
   me.stations[24].raw[46,6] := WSTRING#'';
   me.stations[24].raw[46,7] := WSTRING#'';
   me.stations[24].raw[47,0] := WSTRING#'';
   me.stations[24].raw[47,1] := WSTRING#'';
   me.stations[24].raw[47,2] := WSTRING#'';
   me.stations[24].raw[47,3] := WSTRING#'';
   me.stations[24].raw[47,4] := WSTRING#'';
   me.stations[24].raw[47,5] := WSTRING#'';
   me.stations[24].raw[47,6] := WSTRING#'';
   me.stations[24].raw[47,7] := WSTRING#'';
   me.stations[24].raw[48,0] := WSTRING#'';
   me.stations[24].raw[48,1] := WSTRING#'';
   me.stations[24].raw[48,2] := WSTRING#'';
   me.stations[24].raw[48,3] := WSTRING#'';
   me.stations[24].raw[48,4] := WSTRING#'';
   me.stations[24].raw[48,5] := WSTRING#'';
   me.stations[24].raw[48,6] := WSTRING#'';
   me.stations[24].raw[48,7] := WSTRING#'';
   me.stations[24].raw[49,0] := WSTRING#'';
   me.stations[24].raw[49,1] := WSTRING#'';
   me.stations[24].raw[49,2] := WSTRING#'';
   me.stations[24].raw[49,3] := WSTRING#'';
   me.stations[24].raw[49,4] := WSTRING#'';
   me.stations[24].raw[49,5] := WSTRING#'';
   me.stations[24].raw[49,6] := WSTRING#'';
   me.stations[24].raw[49,7] := WSTRING#'';
   me.stations[25].size := 24;   // cv 01
   me.stations[25].wip[24] := WSTRING#'';   // cv 01
   me.stations[25].wip[25] := WSTRING#'';   // cv 01
   me.stations[25].wip[26] := WSTRING#'';   // cv 01
   me.stations[25].wip[27] := WSTRING#'';   // cv 01
   me.stations[25].wip[28] := WSTRING#'';   // cv 01
   me.stations[25].wip[29] := WSTRING#'';   // cv 01
   me.stations[25].wip[30] := WSTRING#'';   // cv 01
   me.stations[25].wip[31] := WSTRING#'';   // cv 01
   me.stations[25].wip[32] := WSTRING#'';   // cv 01
   me.stations[25].wip[33] := WSTRING#'';   // cv 01
   me.stations[25].wip[34] := WSTRING#'';   // cv 01
   me.stations[25].wip[35] := WSTRING#'';   // cv 01
   me.stations[25].wip[36] := WSTRING#'';   // cv 01
   me.stations[25].wip[37] := WSTRING#'';   // cv 01
   me.stations[25].wip[38] := WSTRING#'';   // cv 01
   me.stations[25].wip[39] := WSTRING#'';   // cv 01
   me.stations[25].wip[40] := WSTRING#'';   // cv 01
   me.stations[25].wip[41] := WSTRING#'';   // cv 01
   me.stations[25].wip[42] := WSTRING#'';   // cv 01
   me.stations[25].wip[43] := WSTRING#'';   // cv 01
   me.stations[25].wip[44] := WSTRING#'';   // cv 01
   me.stations[25].wip[45] := WSTRING#'';   // cv 01
   me.stations[25].wip[46] := WSTRING#'';   // cv 01
   me.stations[25].wip[47] := WSTRING#'';   // cv 01
   me.stations[25].wip[48] := WSTRING#'';   // cv 01
   me.stations[25].wip[49] := WSTRING#'';   // cv 01
   me.stations[25].raw[24,0] := WSTRING#'';   // cv 01
   me.stations[25].raw[24,1] := WSTRING#'';   // cv 01
   me.stations[25].raw[24,2] := WSTRING#'';   // cv 01
   me.stations[25].raw[24,3] := WSTRING#'';   // cv 01
   me.stations[25].raw[24,4] := WSTRING#'';   // cv 01
   me.stations[25].raw[24,5] := WSTRING#'';   // cv 01
   me.stations[25].raw[24,6] := WSTRING#'';   // cv 01
   me.stations[25].raw[24,7] := WSTRING#'';   // cv 01
   me.stations[25].raw[25,0] := WSTRING#'';   // cv 01
   me.stations[25].raw[25,1] := WSTRING#'';   // cv 01
   me.stations[25].raw[25,2] := WSTRING#'';   // cv 01
   me.stations[25].raw[25,3] := WSTRING#'';   // cv 01
   me.stations[25].raw[25,4] := WSTRING#'';   // cv 01
   me.stations[25].raw[25,5] := WSTRING#'';   // cv 01
   me.stations[25].raw[25,6] := WSTRING#'';   // cv 01
   me.stations[25].raw[25,7] := WSTRING#'';   // cv 01
   me.stations[25].raw[26,0] := WSTRING#'';   // cv 01
   me.stations[25].raw[26,1] := WSTRING#'';   // cv 01
   me.stations[25].raw[26,2] := WSTRING#'';   // cv 01
   me.stations[25].raw[26,3] := WSTRING#'';   // cv 01
   me.stations[25].raw[26,4] := WSTRING#'';   // cv 01
   me.stations[25].raw[26,5] := WSTRING#'';   // cv 01
   me.stations[25].raw[26,6] := WSTRING#'';   // cv 01
   me.stations[25].raw[26,7] := WSTRING#'';   // cv 01
   me.stations[25].raw[27,0] := WSTRING#'';   // cv 01
   me.stations[25].raw[27,1] := WSTRING#'';   // cv 01
   me.stations[25].raw[27,2] := WSTRING#'';   // cv 01
   me.stations[25].raw[27,3] := WSTRING#'';   // cv 01
   me.stations[25].raw[27,4] := WSTRING#'';   // cv 01
   me.stations[25].raw[27,5] := WSTRING#'';   // cv 01
   me.stations[25].raw[27,6] := WSTRING#'';   // cv 01
   me.stations[25].raw[27,7] := WSTRING#'';   // cv 01
   me.stations[25].raw[28,0] := WSTRING#'';   // cv 01
   me.stations[25].raw[28,1] := WSTRING#'';   // cv 01
   me.stations[25].raw[28,2] := WSTRING#'';   // cv 01
   me.stations[25].raw[28,3] := WSTRING#'';   // cv 01
   me.stations[25].raw[28,4] := WSTRING#'';   // cv 01
   me.stations[25].raw[28,5] := WSTRING#'';   // cv 01
   me.stations[25].raw[28,6] := WSTRING#'';   // cv 01
   me.stations[25].raw[28,7] := WSTRING#'';   // cv 01
   me.stations[25].raw[29,0] := WSTRING#'';   // cv 01
   me.stations[25].raw[29,1] := WSTRING#'';   // cv 01
   me.stations[25].raw[29,2] := WSTRING#'';   // cv 01
   me.stations[25].raw[29,3] := WSTRING#'';   // cv 01
   me.stations[25].raw[29,4] := WSTRING#'';   // cv 01
   me.stations[25].raw[29,5] := WSTRING#'';   // cv 01
   me.stations[25].raw[29,6] := WSTRING#'';   // cv 01
   me.stations[25].raw[29,7] := WSTRING#'';   // cv 01
   me.stations[25].raw[30,0] := WSTRING#'';   // cv 01
   me.stations[25].raw[30,1] := WSTRING#'';   // cv 01
   me.stations[25].raw[30,2] := WSTRING#'';   // cv 01
   me.stations[25].raw[30,3] := WSTRING#'';   // cv 01
   me.stations[25].raw[30,4] := WSTRING#'';   // cv 01
   me.stations[25].raw[30,5] := WSTRING#'';   // cv 01
   me.stations[25].raw[30,6] := WSTRING#'';   // cv 01
   me.stations[25].raw[30,7] := WSTRING#'';   // cv 01
   me.stations[25].raw[31,0] := WSTRING#'';   // cv 01
   me.stations[25].raw[31,1] := WSTRING#'';   // cv 01
   me.stations[25].raw[31,2] := WSTRING#'';   // cv 01
   me.stations[25].raw[31,3] := WSTRING#'';   // cv 01
   me.stations[25].raw[31,4] := WSTRING#'';   // cv 01
   me.stations[25].raw[31,5] := WSTRING#'';   // cv 01
   me.stations[25].raw[31,6] := WSTRING#'';   // cv 01
   me.stations[25].raw[31,7] := WSTRING#'';   // cv 01
   me.stations[25].raw[32,0] := WSTRING#'';   // cv 01
   me.stations[25].raw[32,1] := WSTRING#'';   // cv 01
   me.stations[25].raw[32,2] := WSTRING#'';   // cv 01
   me.stations[25].raw[32,3] := WSTRING#'';   // cv 01
   me.stations[25].raw[32,4] := WSTRING#'';   // cv 01
   me.stations[25].raw[32,5] := WSTRING#'';   // cv 01
   me.stations[25].raw[32,6] := WSTRING#'';   // cv 01
   me.stations[25].raw[32,7] := WSTRING#'';   // cv 01
   me.stations[25].raw[33,0] := WSTRING#'';   // cv 01
   me.stations[25].raw[33,1] := WSTRING#'';   // cv 01
   me.stations[25].raw[33,2] := WSTRING#'';   // cv 01
   me.stations[25].raw[33,3] := WSTRING#'';   // cv 01
   me.stations[25].raw[33,4] := WSTRING#'';   // cv 01
   me.stations[25].raw[33,5] := WSTRING#'';   // cv 01
   me.stations[25].raw[33,6] := WSTRING#'';   // cv 01
   me.stations[25].raw[33,7] := WSTRING#'';   // cv 01
   me.stations[25].raw[34,0] := WSTRING#'';   // cv 01
   me.stations[25].raw[34,1] := WSTRING#'';   // cv 01
   me.stations[25].raw[34,2] := WSTRING#'';   // cv 01
   me.stations[25].raw[34,3] := WSTRING#'';   // cv 01
   me.stations[25].raw[34,4] := WSTRING#'';   // cv 01
   me.stations[25].raw[34,5] := WSTRING#'';   // cv 01
   me.stations[25].raw[34,6] := WSTRING#'';   // cv 01
   me.stations[25].raw[34,7] := WSTRING#'';   // cv 01
   me.stations[25].raw[35,0] := WSTRING#'';   // cv 01
   me.stations[25].raw[35,1] := WSTRING#'';   // cv 01
   me.stations[25].raw[35,2] := WSTRING#'';   // cv 01
   me.stations[25].raw[35,3] := WSTRING#'';   // cv 01
   me.stations[25].raw[35,4] := WSTRING#'';   // cv 01
   me.stations[25].raw[35,5] := WSTRING#'';   // cv 01
   me.stations[25].raw[35,6] := WSTRING#'';   // cv 01
   me.stations[25].raw[35,7] := WSTRING#'';   // cv 01
   me.stations[25].raw[36,0] := WSTRING#'';   // cv 01
   me.stations[25].raw[36,1] := WSTRING#'';   // cv 01
   me.stations[25].raw[36,2] := WSTRING#'';   // cv 01
   me.stations[25].raw[36,3] := WSTRING#'';   // cv 01
   me.stations[25].raw[36,4] := WSTRING#'';   // cv 01
   me.stations[25].raw[36,5] := WSTRING#'';   // cv 01
   me.stations[25].raw[36,6] := WSTRING#'';   // cv 01
   me.stations[25].raw[36,7] := WSTRING#'';   // cv 01
   me.stations[25].raw[37,0] := WSTRING#'';   // cv 01
   me.stations[25].raw[37,1] := WSTRING#'';   // cv 01
   me.stations[25].raw[37,2] := WSTRING#'';   // cv 01
   me.stations[25].raw[37,3] := WSTRING#'';   // cv 01
   me.stations[25].raw[37,4] := WSTRING#'';   // cv 01
   me.stations[25].raw[37,5] := WSTRING#'';   // cv 01
   me.stations[25].raw[37,6] := WSTRING#'';   // cv 01
   me.stations[25].raw[37,7] := WSTRING#'';   // cv 01
   me.stations[25].raw[38,0] := WSTRING#'';   // cv 01
   me.stations[25].raw[38,1] := WSTRING#'';   // cv 01
   me.stations[25].raw[38,2] := WSTRING#'';   // cv 01
   me.stations[25].raw[38,3] := WSTRING#'';   // cv 01
   me.stations[25].raw[38,4] := WSTRING#'';   // cv 01
   me.stations[25].raw[38,5] := WSTRING#'';   // cv 01
   me.stations[25].raw[38,6] := WSTRING#'';   // cv 01
   me.stations[25].raw[38,7] := WSTRING#'';   // cv 01
   me.stations[25].raw[39,0] := WSTRING#'';   // cv 01
   me.stations[25].raw[39,1] := WSTRING#'';   // cv 01
   me.stations[25].raw[39,2] := WSTRING#'';   // cv 01
   me.stations[25].raw[39,3] := WSTRING#'';   // cv 01
   me.stations[25].raw[39,4] := WSTRING#'';   // cv 01
   me.stations[25].raw[39,5] := WSTRING#'';   // cv 01
   me.stations[25].raw[39,6] := WSTRING#'';   // cv 01
   me.stations[25].raw[39,7] := WSTRING#'';   // cv 01
   me.stations[25].raw[40,0] := WSTRING#'';   // cv 01
   me.stations[25].raw[40,1] := WSTRING#'';   // cv 01
   me.stations[25].raw[40,2] := WSTRING#'';   // cv 01
   me.stations[25].raw[40,3] := WSTRING#'';   // cv 01
   me.stations[25].raw[40,4] := WSTRING#'';   // cv 01
   me.stations[25].raw[40,5] := WSTRING#'';   // cv 01
   me.stations[25].raw[40,6] := WSTRING#'';   // cv 01
   me.stations[25].raw[40,7] := WSTRING#'';   // cv 01
   me.stations[25].raw[41,0] := WSTRING#'';   // cv 01
   me.stations[25].raw[41,1] := WSTRING#'';   // cv 01
   me.stations[25].raw[41,2] := WSTRING#'';   // cv 01
   me.stations[25].raw[41,3] := WSTRING#'';   // cv 01
   me.stations[25].raw[41,4] := WSTRING#'';   // cv 01
   me.stations[25].raw[41,5] := WSTRING#'';   // cv 01
   me.stations[25].raw[41,6] := WSTRING#'';   // cv 01
   me.stations[25].raw[41,7] := WSTRING#'';   // cv 01
   me.stations[25].raw[42,0] := WSTRING#'';   // cv 01
   me.stations[25].raw[42,1] := WSTRING#'';   // cv 01
   me.stations[25].raw[42,2] := WSTRING#'';   // cv 01
   me.stations[25].raw[42,3] := WSTRING#'';   // cv 01
   me.stations[25].raw[42,4] := WSTRING#'';   // cv 01
   me.stations[25].raw[42,5] := WSTRING#'';   // cv 01
   me.stations[25].raw[42,6] := WSTRING#'';   // cv 01
   me.stations[25].raw[42,7] := WSTRING#'';   // cv 01
   me.stations[25].raw[43,0] := WSTRING#'';   // cv 01
   me.stations[25].raw[43,1] := WSTRING#'';   // cv 01
   me.stations[25].raw[43,2] := WSTRING#'';   // cv 01
   me.stations[25].raw[43,3] := WSTRING#'';   // cv 01
   me.stations[25].raw[43,4] := WSTRING#'';   // cv 01
   me.stations[25].raw[43,5] := WSTRING#'';   // cv 01
   me.stations[25].raw[43,6] := WSTRING#'';   // cv 01
   me.stations[25].raw[43,7] := WSTRING#'';   // cv 01
   me.stations[25].raw[44,0] := WSTRING#'';   // cv 01
   me.stations[25].raw[44,1] := WSTRING#'';   // cv 01
   me.stations[25].raw[44,2] := WSTRING#'';   // cv 01
   me.stations[25].raw[44,3] := WSTRING#'';   // cv 01
   me.stations[25].raw[44,4] := WSTRING#'';   // cv 01
   me.stations[25].raw[44,5] := WSTRING#'';   // cv 01
   me.stations[25].raw[44,6] := WSTRING#'';   // cv 01
   me.stations[25].raw[44,7] := WSTRING#'';   // cv 01
   me.stations[25].raw[45,0] := WSTRING#'';   // cv 01
   me.stations[25].raw[45,1] := WSTRING#'';   // cv 01
   me.stations[25].raw[45,2] := WSTRING#'';   // cv 01
   me.stations[25].raw[45,3] := WSTRING#'';   // cv 01
   me.stations[25].raw[45,4] := WSTRING#'';   // cv 01
   me.stations[25].raw[45,5] := WSTRING#'';   // cv 01
   me.stations[25].raw[45,6] := WSTRING#'';   // cv 01
   me.stations[25].raw[45,7] := WSTRING#'';   // cv 01
   me.stations[25].raw[46,0] := WSTRING#'';   // cv 01
   me.stations[25].raw[46,1] := WSTRING#'';   // cv 01
   me.stations[25].raw[46,2] := WSTRING#'';   // cv 01
   me.stations[25].raw[46,3] := WSTRING#'';   // cv 01
   me.stations[25].raw[46,4] := WSTRING#'';   // cv 01
   me.stations[25].raw[46,5] := WSTRING#'';   // cv 01
   me.stations[25].raw[46,6] := WSTRING#'';   // cv 01
   me.stations[25].raw[46,7] := WSTRING#'';   // cv 01
   me.stations[25].raw[47,0] := WSTRING#'';   // cv 01
   me.stations[25].raw[47,1] := WSTRING#'';   // cv 01
   me.stations[25].raw[47,2] := WSTRING#'';   // cv 01
   me.stations[25].raw[47,3] := WSTRING#'';   // cv 01
   me.stations[25].raw[47,4] := WSTRING#'';   // cv 01
   me.stations[25].raw[47,5] := WSTRING#'';   // cv 01
   me.stations[25].raw[47,6] := WSTRING#'';   // cv 01
   me.stations[25].raw[47,7] := WSTRING#'';   // cv 01
   me.stations[25].raw[48,0] := WSTRING#'';   // cv 01
   me.stations[25].raw[48,1] := WSTRING#'';   // cv 01
   me.stations[25].raw[48,2] := WSTRING#'';   // cv 01
   me.stations[25].raw[48,3] := WSTRING#'';   // cv 01
   me.stations[25].raw[48,4] := WSTRING#'';   // cv 01
   me.stations[25].raw[48,5] := WSTRING#'';   // cv 01
   me.stations[25].raw[48,6] := WSTRING#'';   // cv 01
   me.stations[25].raw[48,7] := WSTRING#'';   // cv 01
   me.stations[25].raw[49,0] := WSTRING#'';   // cv 01
   me.stations[25].raw[49,1] := WSTRING#'';   // cv 01
   me.stations[25].raw[49,2] := WSTRING#'';   // cv 01
   me.stations[25].raw[49,3] := WSTRING#'';   // cv 01
   me.stations[25].raw[49,4] := WSTRING#'';   // cv 01
   me.stations[25].raw[49,5] := WSTRING#'';   // cv 01
   me.stations[25].raw[49,6] := WSTRING#'';   // cv 01
   me.stations[25].raw[49,7] := WSTRING#'';   // cv 01
   me.stations[26].size := 14;   // cv 02
   me.stations[26].wip[13] := WSTRING#'16.08.216.751.100A$LSA Sleeved SCR 2016';   // cv 02
   me.stations[26].wip[14] := WSTRING#'';   // cv 02
   me.stations[26].wip[15] := WSTRING#'';   // cv 02
   me.stations[26].wip[16] := WSTRING#'';   // cv 02
   me.stations[26].wip[17] := WSTRING#'';   // cv 02
   me.stations[26].wip[18] := WSTRING#'';   // cv 02
   me.stations[26].wip[19] := WSTRING#'';   // cv 02
   me.stations[26].wip[20] := WSTRING#'';   // cv 02
   me.stations[26].wip[21] := WSTRING#'';   // cv 02
   me.stations[26].wip[22] := WSTRING#'';   // cv 02
   me.stations[26].wip[23] := WSTRING#'';   // cv 02
   me.stations[26].wip[24] := WSTRING#'';   // cv 02
   me.stations[26].wip[25] := WSTRING#'';   // cv 02
   me.stations[26].wip[26] := WSTRING#'';   // cv 02
   me.stations[26].wip[27] := WSTRING#'';   // cv 02
   me.stations[26].wip[28] := WSTRING#'';   // cv 02
   me.stations[26].wip[29] := WSTRING#'';   // cv 02
   me.stations[26].wip[30] := WSTRING#'';   // cv 02
   me.stations[26].wip[31] := WSTRING#'';   // cv 02
   me.stations[26].wip[32] := WSTRING#'';   // cv 02
   me.stations[26].wip[33] := WSTRING#'';   // cv 02
   me.stations[26].wip[34] := WSTRING#'';   // cv 02
   me.stations[26].wip[35] := WSTRING#'';   // cv 02
   me.stations[26].wip[36] := WSTRING#'';   // cv 02
   me.stations[26].wip[37] := WSTRING#'';   // cv 02
   me.stations[26].wip[38] := WSTRING#'';   // cv 02
   me.stations[26].wip[39] := WSTRING#'';   // cv 02
   me.stations[26].wip[40] := WSTRING#'';   // cv 02
   me.stations[26].wip[41] := WSTRING#'';   // cv 02
   me.stations[26].wip[42] := WSTRING#'';   // cv 02
   me.stations[26].wip[43] := WSTRING#'';   // cv 02
   me.stations[26].wip[44] := WSTRING#'';   // cv 02
   me.stations[26].wip[45] := WSTRING#'';   // cv 02
   me.stations[26].wip[46] := WSTRING#'';   // cv 02
   me.stations[26].wip[47] := WSTRING#'';   // cv 02
   me.stations[26].wip[48] := WSTRING#'';   // cv 02
   me.stations[26].wip[49] := WSTRING#'';   // cv 02
   me.stations[26].raw[13,0] := WSTRING#'';   // cv 02
   me.stations[26].raw[13,1] := WSTRING#'C/O MATERIALS';   // cv 02
   me.stations[26].raw[13,2] := WSTRING#'16.08.216.291.000A';   // cv 02
   me.stations[26].raw[13,3] := WSTRING#'16.08.216.315.001A';   // cv 02
   me.stations[26].raw[13,4] := WSTRING#'';   // cv 02
   me.stations[26].raw[13,5] := WSTRING#'16.08.216.057.001A';   // cv 02
   me.stations[26].raw[13,6] := WSTRING#'16.08.208.661.000F';   // cv 02
   me.stations[26].raw[13,7] := WSTRING#'16.08.216.315.002A';   // cv 02
   me.stations[26].raw[14,0] := WSTRING#'';   // cv 02
   me.stations[26].raw[14,1] := WSTRING#'';   // cv 02
   me.stations[26].raw[14,2] := WSTRING#'';   // cv 02
   me.stations[26].raw[14,3] := WSTRING#'';   // cv 02
   me.stations[26].raw[14,4] := WSTRING#'';   // cv 02
   me.stations[26].raw[14,5] := WSTRING#'';   // cv 02
   me.stations[26].raw[14,6] := WSTRING#'';   // cv 02
   me.stations[26].raw[14,7] := WSTRING#'';   // cv 02
   me.stations[26].raw[15,0] := WSTRING#'';   // cv 02
   me.stations[26].raw[15,1] := WSTRING#'';   // cv 02
   me.stations[26].raw[15,2] := WSTRING#'';   // cv 02
   me.stations[26].raw[15,3] := WSTRING#'';   // cv 02
   me.stations[26].raw[15,4] := WSTRING#'';   // cv 02
   me.stations[26].raw[15,5] := WSTRING#'';   // cv 02
   me.stations[26].raw[15,6] := WSTRING#'';   // cv 02
   me.stations[26].raw[15,7] := WSTRING#'';   // cv 02
   me.stations[26].raw[16,0] := WSTRING#'';   // cv 02
   me.stations[26].raw[16,1] := WSTRING#'';   // cv 02
   me.stations[26].raw[16,2] := WSTRING#'';   // cv 02
   me.stations[26].raw[16,3] := WSTRING#'';   // cv 02
   me.stations[26].raw[16,4] := WSTRING#'';   // cv 02
   me.stations[26].raw[16,5] := WSTRING#'';   // cv 02
   me.stations[26].raw[16,6] := WSTRING#'';   // cv 02
   me.stations[26].raw[16,7] := WSTRING#'';   // cv 02
   me.stations[26].raw[17,0] := WSTRING#'';   // cv 02
   me.stations[26].raw[17,1] := WSTRING#'';   // cv 02
   me.stations[26].raw[17,2] := WSTRING#'';   // cv 02
   me.stations[26].raw[17,3] := WSTRING#'';   // cv 02
   me.stations[26].raw[17,4] := WSTRING#'';   // cv 02
   me.stations[26].raw[17,5] := WSTRING#'';   // cv 02
   me.stations[26].raw[17,6] := WSTRING#'';   // cv 02
   me.stations[26].raw[17,7] := WSTRING#'';   // cv 02
   me.stations[26].raw[18,0] := WSTRING#'';   // cv 02
   me.stations[26].raw[18,1] := WSTRING#'';   // cv 02
   me.stations[26].raw[18,2] := WSTRING#'';   // cv 02
   me.stations[26].raw[18,3] := WSTRING#'';   // cv 02
   me.stations[26].raw[18,4] := WSTRING#'';   // cv 02
   me.stations[26].raw[18,5] := WSTRING#'';   // cv 02
   me.stations[26].raw[18,6] := WSTRING#'';   // cv 02
   me.stations[26].raw[18,7] := WSTRING#'';   // cv 02
   me.stations[26].raw[19,0] := WSTRING#'';   // cv 02
   me.stations[26].raw[19,1] := WSTRING#'';   // cv 02
   me.stations[26].raw[19,2] := WSTRING#'';   // cv 02
   me.stations[26].raw[19,3] := WSTRING#'';   // cv 02
   me.stations[26].raw[19,4] := WSTRING#'';   // cv 02
   me.stations[26].raw[19,5] := WSTRING#'';   // cv 02
   me.stations[26].raw[19,6] := WSTRING#'';   // cv 02
   me.stations[26].raw[19,7] := WSTRING#'';   // cv 02
   me.stations[26].raw[20,0] := WSTRING#'';   // cv 02
   me.stations[26].raw[20,1] := WSTRING#'';   // cv 02
   me.stations[26].raw[20,2] := WSTRING#'';   // cv 02
   me.stations[26].raw[20,3] := WSTRING#'';   // cv 02
   me.stations[26].raw[20,4] := WSTRING#'';   // cv 02
   me.stations[26].raw[20,5] := WSTRING#'';   // cv 02
   me.stations[26].raw[20,6] := WSTRING#'';   // cv 02
   me.stations[26].raw[20,7] := WSTRING#'';   // cv 02
   me.stations[26].raw[21,0] := WSTRING#'';   // cv 02
   me.stations[26].raw[21,1] := WSTRING#'';   // cv 02
   me.stations[26].raw[21,2] := WSTRING#'';   // cv 02
   me.stations[26].raw[21,3] := WSTRING#'';   // cv 02
   me.stations[26].raw[21,4] := WSTRING#'';   // cv 02
   me.stations[26].raw[21,5] := WSTRING#'';   // cv 02
   me.stations[26].raw[21,6] := WSTRING#'';   // cv 02
   me.stations[26].raw[21,7] := WSTRING#'';   // cv 02
   me.stations[26].raw[22,0] := WSTRING#'';   // cv 02
   me.stations[26].raw[22,1] := WSTRING#'';   // cv 02
   me.stations[26].raw[22,2] := WSTRING#'';   // cv 02
   me.stations[26].raw[22,3] := WSTRING#'';   // cv 02
   me.stations[26].raw[22,4] := WSTRING#'';   // cv 02
   me.stations[26].raw[22,5] := WSTRING#'';   // cv 02
   me.stations[26].raw[22,6] := WSTRING#'';   // cv 02
   me.stations[26].raw[22,7] := WSTRING#'';   // cv 02
   me.stations[26].raw[23,0] := WSTRING#'';   // cv 02
   me.stations[26].raw[23,1] := WSTRING#'';   // cv 02
   me.stations[26].raw[23,2] := WSTRING#'';   // cv 02
   me.stations[26].raw[23,3] := WSTRING#'';   // cv 02
   me.stations[26].raw[23,4] := WSTRING#'';   // cv 02
   me.stations[26].raw[23,5] := WSTRING#'';   // cv 02
   me.stations[26].raw[23,6] := WSTRING#'';   // cv 02
   me.stations[26].raw[23,7] := WSTRING#'';   // cv 02
   me.stations[26].raw[24,0] := WSTRING#'';   // cv 02
   me.stations[26].raw[24,1] := WSTRING#'';   // cv 02
   me.stations[26].raw[24,2] := WSTRING#'';   // cv 02
   me.stations[26].raw[24,3] := WSTRING#'';   // cv 02
   me.stations[26].raw[24,4] := WSTRING#'';   // cv 02
   me.stations[26].raw[24,5] := WSTRING#'';   // cv 02
   me.stations[26].raw[24,6] := WSTRING#'';   // cv 02
   me.stations[26].raw[24,7] := WSTRING#'';   // cv 02
   me.stations[26].raw[25,0] := WSTRING#'';   // cv 02
   me.stations[26].raw[25,1] := WSTRING#'';   // cv 02
   me.stations[26].raw[25,2] := WSTRING#'';   // cv 02
   me.stations[26].raw[25,3] := WSTRING#'';   // cv 02
   me.stations[26].raw[25,4] := WSTRING#'';   // cv 02
   me.stations[26].raw[25,5] := WSTRING#'';   // cv 02
   me.stations[26].raw[25,6] := WSTRING#'';   // cv 02
   me.stations[26].raw[25,7] := WSTRING#'';   // cv 02
   me.stations[26].raw[26,0] := WSTRING#'';   // cv 02
   me.stations[26].raw[26,1] := WSTRING#'';   // cv 02
   me.stations[26].raw[26,2] := WSTRING#'';   // cv 02
   me.stations[26].raw[26,3] := WSTRING#'';   // cv 02
   me.stations[26].raw[26,4] := WSTRING#'';   // cv 02
   me.stations[26].raw[26,5] := WSTRING#'';   // cv 02
   me.stations[26].raw[26,6] := WSTRING#'';   // cv 02
   me.stations[26].raw[26,7] := WSTRING#'';   // cv 02
   me.stations[26].raw[27,0] := WSTRING#'';   // cv 02
   me.stations[26].raw[27,1] := WSTRING#'';   // cv 02
   me.stations[26].raw[27,2] := WSTRING#'';   // cv 02
   me.stations[26].raw[27,3] := WSTRING#'';   // cv 02
   me.stations[26].raw[27,4] := WSTRING#'';   // cv 02
   me.stations[26].raw[27,5] := WSTRING#'';   // cv 02
   me.stations[26].raw[27,6] := WSTRING#'';   // cv 02
   me.stations[26].raw[27,7] := WSTRING#'';   // cv 02
   me.stations[26].raw[28,0] := WSTRING#'';   // cv 02
   me.stations[26].raw[28,1] := WSTRING#'';   // cv 02
   me.stations[26].raw[28,2] := WSTRING#'';   // cv 02
   me.stations[26].raw[28,3] := WSTRING#'';   // cv 02
   me.stations[26].raw[28,4] := WSTRING#'';   // cv 02
   me.stations[26].raw[28,5] := WSTRING#'';   // cv 02
   me.stations[26].raw[28,6] := WSTRING#'';   // cv 02
   me.stations[26].raw[28,7] := WSTRING#'';   // cv 02
   me.stations[26].raw[29,0] := WSTRING#'';   // cv 02
   me.stations[26].raw[29,1] := WSTRING#'';   // cv 02
   me.stations[26].raw[29,2] := WSTRING#'';   // cv 02
   me.stations[26].raw[29,3] := WSTRING#'';   // cv 02
   me.stations[26].raw[29,4] := WSTRING#'';   // cv 02
   me.stations[26].raw[29,5] := WSTRING#'';   // cv 02
   me.stations[26].raw[29,6] := WSTRING#'';   // cv 02
   me.stations[26].raw[29,7] := WSTRING#'';   // cv 02
   me.stations[26].raw[30,0] := WSTRING#'';   // cv 02
   me.stations[26].raw[30,1] := WSTRING#'';   // cv 02
   me.stations[26].raw[30,2] := WSTRING#'';   // cv 02
   me.stations[26].raw[30,3] := WSTRING#'';   // cv 02
   me.stations[26].raw[30,4] := WSTRING#'';   // cv 02
   me.stations[26].raw[30,5] := WSTRING#'';   // cv 02
   me.stations[26].raw[30,6] := WSTRING#'';   // cv 02
   me.stations[26].raw[30,7] := WSTRING#'';   // cv 02
   me.stations[26].raw[31,0] := WSTRING#'';   // cv 02
   me.stations[26].raw[31,1] := WSTRING#'';   // cv 02
   me.stations[26].raw[31,2] := WSTRING#'';   // cv 02
   me.stations[26].raw[31,3] := WSTRING#'';   // cv 02
   me.stations[26].raw[31,4] := WSTRING#'';   // cv 02
   me.stations[26].raw[31,5] := WSTRING#'';   // cv 02
   me.stations[26].raw[31,6] := WSTRING#'';   // cv 02
   me.stations[26].raw[31,7] := WSTRING#'';   // cv 02
   me.stations[26].raw[32,0] := WSTRING#'';   // cv 02
   me.stations[26].raw[32,1] := WSTRING#'';   // cv 02
   me.stations[26].raw[32,2] := WSTRING#'';   // cv 02
   me.stations[26].raw[32,3] := WSTRING#'';   // cv 02
   me.stations[26].raw[32,4] := WSTRING#'';   // cv 02
   me.stations[26].raw[32,5] := WSTRING#'';   // cv 02
   me.stations[26].raw[32,6] := WSTRING#'';   // cv 02
   me.stations[26].raw[32,7] := WSTRING#'';   // cv 02
   me.stations[26].raw[33,0] := WSTRING#'';   // cv 02
   me.stations[26].raw[33,1] := WSTRING#'';   // cv 02
   me.stations[26].raw[33,2] := WSTRING#'';   // cv 02
   me.stations[26].raw[33,3] := WSTRING#'';   // cv 02
   me.stations[26].raw[33,4] := WSTRING#'';   // cv 02
   me.stations[26].raw[33,5] := WSTRING#'';   // cv 02
   me.stations[26].raw[33,6] := WSTRING#'';   // cv 02
   me.stations[26].raw[33,7] := WSTRING#'';   // cv 02
   me.stations[26].raw[34,0] := WSTRING#'';   // cv 02
   me.stations[26].raw[34,1] := WSTRING#'';   // cv 02
   me.stations[26].raw[34,2] := WSTRING#'';   // cv 02
   me.stations[26].raw[34,3] := WSTRING#'';   // cv 02
   me.stations[26].raw[34,4] := WSTRING#'';   // cv 02
   me.stations[26].raw[34,5] := WSTRING#'';   // cv 02
   me.stations[26].raw[34,6] := WSTRING#'';   // cv 02
   me.stations[26].raw[34,7] := WSTRING#'';   // cv 02
   me.stations[26].raw[35,0] := WSTRING#'';   // cv 02
   me.stations[26].raw[35,1] := WSTRING#'';   // cv 02
   me.stations[26].raw[35,2] := WSTRING#'';   // cv 02
   me.stations[26].raw[35,3] := WSTRING#'';   // cv 02
   me.stations[26].raw[35,4] := WSTRING#'';   // cv 02
   me.stations[26].raw[35,5] := WSTRING#'';   // cv 02
   me.stations[26].raw[35,6] := WSTRING#'';   // cv 02
   me.stations[26].raw[35,7] := WSTRING#'';   // cv 02
   me.stations[26].raw[36,0] := WSTRING#'';   // cv 02
   me.stations[26].raw[36,1] := WSTRING#'';   // cv 02
   me.stations[26].raw[36,2] := WSTRING#'';   // cv 02
   me.stations[26].raw[36,3] := WSTRING#'';   // cv 02
   me.stations[26].raw[36,4] := WSTRING#'';   // cv 02
   me.stations[26].raw[36,5] := WSTRING#'';   // cv 02
   me.stations[26].raw[36,6] := WSTRING#'';   // cv 02
   me.stations[26].raw[36,7] := WSTRING#'';   // cv 02
   me.stations[26].raw[37,0] := WSTRING#'';   // cv 02
   me.stations[26].raw[37,1] := WSTRING#'';   // cv 02
   me.stations[26].raw[37,2] := WSTRING#'';   // cv 02
   me.stations[26].raw[37,3] := WSTRING#'';   // cv 02
   me.stations[26].raw[37,4] := WSTRING#'';   // cv 02
   me.stations[26].raw[37,5] := WSTRING#'';   // cv 02
   me.stations[26].raw[37,6] := WSTRING#'';   // cv 02
   me.stations[26].raw[37,7] := WSTRING#'';   // cv 02
   me.stations[26].raw[38,0] := WSTRING#'';   // cv 02
   me.stations[26].raw[38,1] := WSTRING#'';   // cv 02
   me.stations[26].raw[38,2] := WSTRING#'';   // cv 02
   me.stations[26].raw[38,3] := WSTRING#'';   // cv 02
   me.stations[26].raw[38,4] := WSTRING#'';   // cv 02
   me.stations[26].raw[38,5] := WSTRING#'';   // cv 02
   me.stations[26].raw[38,6] := WSTRING#'';   // cv 02
   me.stations[26].raw[38,7] := WSTRING#'';   // cv 02
   me.stations[26].raw[39,0] := WSTRING#'';   // cv 02
   me.stations[26].raw[39,1] := WSTRING#'';   // cv 02
   me.stations[26].raw[39,2] := WSTRING#'';   // cv 02
   me.stations[26].raw[39,3] := WSTRING#'';   // cv 02
   me.stations[26].raw[39,4] := WSTRING#'';   // cv 02
   me.stations[26].raw[39,5] := WSTRING#'';   // cv 02
   me.stations[26].raw[39,6] := WSTRING#'';   // cv 02
   me.stations[26].raw[39,7] := WSTRING#'';   // cv 02
   me.stations[26].raw[40,0] := WSTRING#'';   // cv 02
   me.stations[26].raw[40,1] := WSTRING#'';   // cv 02
   me.stations[26].raw[40,2] := WSTRING#'';   // cv 02
   me.stations[26].raw[40,3] := WSTRING#'';   // cv 02
   me.stations[26].raw[40,4] := WSTRING#'';   // cv 02
   me.stations[26].raw[40,5] := WSTRING#'';   // cv 02
   me.stations[26].raw[40,6] := WSTRING#'';   // cv 02
   me.stations[26].raw[40,7] := WSTRING#'';   // cv 02
   me.stations[26].raw[41,0] := WSTRING#'';   // cv 02
   me.stations[26].raw[41,1] := WSTRING#'';   // cv 02
   me.stations[26].raw[41,2] := WSTRING#'';   // cv 02
   me.stations[26].raw[41,3] := WSTRING#'';   // cv 02
   me.stations[26].raw[41,4] := WSTRING#'';   // cv 02
   me.stations[26].raw[41,5] := WSTRING#'';   // cv 02
   me.stations[26].raw[41,6] := WSTRING#'';   // cv 02
   me.stations[26].raw[41,7] := WSTRING#'';   // cv 02
   me.stations[26].raw[42,0] := WSTRING#'';   // cv 02
   me.stations[26].raw[42,1] := WSTRING#'';   // cv 02
   me.stations[26].raw[42,2] := WSTRING#'';   // cv 02
   me.stations[26].raw[42,3] := WSTRING#'';   // cv 02
   me.stations[26].raw[42,4] := WSTRING#'';   // cv 02
   me.stations[26].raw[42,5] := WSTRING#'';   // cv 02
   me.stations[26].raw[42,6] := WSTRING#'';   // cv 02
   me.stations[26].raw[42,7] := WSTRING#'';   // cv 02
   me.stations[26].raw[43,0] := WSTRING#'';   // cv 02
   me.stations[26].raw[43,1] := WSTRING#'';   // cv 02
   me.stations[26].raw[43,2] := WSTRING#'';   // cv 02
   me.stations[26].raw[43,3] := WSTRING#'';   // cv 02
   me.stations[26].raw[43,4] := WSTRING#'';   // cv 02
   me.stations[26].raw[43,5] := WSTRING#'';   // cv 02
   me.stations[26].raw[43,6] := WSTRING#'';   // cv 02
   me.stations[26].raw[43,7] := WSTRING#'';   // cv 02
   me.stations[26].raw[44,0] := WSTRING#'';   // cv 02
   me.stations[26].raw[44,1] := WSTRING#'';   // cv 02
   me.stations[26].raw[44,2] := WSTRING#'';   // cv 02
   me.stations[26].raw[44,3] := WSTRING#'';   // cv 02
   me.stations[26].raw[44,4] := WSTRING#'';   // cv 02
   me.stations[26].raw[44,5] := WSTRING#'';   // cv 02
   me.stations[26].raw[44,6] := WSTRING#'';   // cv 02
   me.stations[26].raw[44,7] := WSTRING#'';   // cv 02
   me.stations[26].raw[45,0] := WSTRING#'';   // cv 02
   me.stations[26].raw[45,1] := WSTRING#'';   // cv 02
   me.stations[26].raw[45,2] := WSTRING#'';   // cv 02
   me.stations[26].raw[45,3] := WSTRING#'';   // cv 02
   me.stations[26].raw[45,4] := WSTRING#'';   // cv 02
   me.stations[26].raw[45,5] := WSTRING#'';   // cv 02
   me.stations[26].raw[45,6] := WSTRING#'';   // cv 02
   me.stations[26].raw[45,7] := WSTRING#'';   // cv 02
   me.stations[26].raw[46,0] := WSTRING#'';   // cv 02
   me.stations[26].raw[46,1] := WSTRING#'';   // cv 02
   me.stations[26].raw[46,2] := WSTRING#'';   // cv 02
   me.stations[26].raw[46,3] := WSTRING#'';   // cv 02
   me.stations[26].raw[46,4] := WSTRING#'';   // cv 02
   me.stations[26].raw[46,5] := WSTRING#'';   // cv 02
   me.stations[26].raw[46,6] := WSTRING#'';   // cv 02
   me.stations[26].raw[46,7] := WSTRING#'';   // cv 02
   me.stations[26].raw[47,0] := WSTRING#'';   // cv 02
   me.stations[26].raw[47,1] := WSTRING#'';   // cv 02
   me.stations[26].raw[47,2] := WSTRING#'';   // cv 02
   me.stations[26].raw[47,3] := WSTRING#'';   // cv 02
   me.stations[26].raw[47,4] := WSTRING#'';   // cv 02
   me.stations[26].raw[47,5] := WSTRING#'';   // cv 02
   me.stations[26].raw[47,6] := WSTRING#'';   // cv 02
   me.stations[26].raw[47,7] := WSTRING#'';   // cv 02
   me.stations[26].raw[48,0] := WSTRING#'';   // cv 02
   me.stations[26].raw[48,1] := WSTRING#'';   // cv 02
   me.stations[26].raw[48,2] := WSTRING#'';   // cv 02
   me.stations[26].raw[48,3] := WSTRING#'';   // cv 02
   me.stations[26].raw[48,4] := WSTRING#'';   // cv 02
   me.stations[26].raw[48,5] := WSTRING#'';   // cv 02
   me.stations[26].raw[48,6] := WSTRING#'';   // cv 02
   me.stations[26].raw[48,7] := WSTRING#'';   // cv 02
   me.stations[26].raw[49,0] := WSTRING#'';   // cv 02
   me.stations[26].raw[49,1] := WSTRING#'';   // cv 02
   me.stations[26].raw[49,2] := WSTRING#'';   // cv 02
   me.stations[26].raw[49,3] := WSTRING#'';   // cv 02
   me.stations[26].raw[49,4] := WSTRING#'';   // cv 02
   me.stations[26].raw[49,5] := WSTRING#'';   // cv 02
   me.stations[26].raw[49,6] := WSTRING#'';   // cv 02
   me.stations[26].raw[49,7] := WSTRING#'';   // cv 02
   me.stations[27].size := 46;   // cv 03
   me.stations[27].wip[41] := WSTRING#'16.32.606.411.000A$LStuffed Shell - SCR Horizontal';   // cv 03
   me.stations[27].wip[42] := WSTRING#'16.32.112.304.008A$LASSY SCR CANNING FORMED';   // cv 03
   me.stations[27].wip[43] := WSTRING#'16.08.211.806.400B$LSA DPF Stuffed Shell';   // cv 03
   me.stations[27].wip[44] := WSTRING#'16.08.208.651.000G$LStuffed Shell SCR- NGK';   // cv 03
   me.stations[27].wip[45] := WSTRING#'16.18.008.330.000A';   // cv 03
   me.stations[27].wip[46] := WSTRING#'';   // cv 03
   me.stations[27].wip[47] := WSTRING#'';   // cv 03
   me.stations[27].wip[48] := WSTRING#'';   // cv 03
   me.stations[27].wip[49] := WSTRING#'';   // cv 03
   me.stations[27].raw[41,0] := WSTRING#'';   // cv 03
   me.stations[27].raw[41,1] := WSTRING#'FINISHED GOODS';   // cv 03
   me.stations[27].raw[41,2] := WSTRING#'16.32.606.311.040B';   // cv 03
   me.stations[27].raw[41,3] := WSTRING#'16.32.606.311.070A';   // cv 03
   me.stations[27].raw[41,4] := WSTRING#'';   // cv 03
   me.stations[27].raw[41,5] := WSTRING#'16.32.606.311.050B';   // cv 03
   me.stations[27].raw[41,6] := WSTRING#'16.32.606.311.010F';   // cv 03
   me.stations[27].raw[41,7] := WSTRING#'16.32.606.311.060A';   // cv 03
   me.stations[27].raw[42,0] := WSTRING#'';   // cv 03
   me.stations[27].raw[42,1] := WSTRING#'FINISHED GOODS';   // cv 03
   me.stations[27].raw[42,2] := WSTRING#'16.32.112.054.041A';   // cv 03
   me.stations[27].raw[42,3] := WSTRING#'';   // cv 03
   me.stations[27].raw[42,4] := WSTRING#'';   // cv 03
   me.stations[27].raw[42,5] := WSTRING#'16.32.112.057.010A';   // cv 03
   me.stations[27].raw[42,6] := WSTRING#'16.32.112.553.100D';   // cv 03
   me.stations[27].raw[42,7] := WSTRING#'16.32.806.315.001A';   // cv 03
   me.stations[27].raw[43,0] := WSTRING#'';   // cv 03
   me.stations[27].raw[43,1] := WSTRING#'FINISHED GOODS';   // cv 03
   me.stations[27].raw[43,2] := WSTRING#'16.08.211.806.020A';   // cv 03
   me.stations[27].raw[43,3] := WSTRING#'';   // cv 03
   me.stations[27].raw[43,4] := WSTRING#'';   // cv 03
   me.stations[27].raw[43,5] := WSTRING#'';   // cv 03
   me.stations[27].raw[43,6] := WSTRING#'16.08.208.631.000F';   // cv 03
   me.stations[27].raw[43,7] := WSTRING#'16.08.216.315.000A';   // cv 03
   me.stations[27].raw[44,0] := WSTRING#'';   // cv 03
   me.stations[27].raw[44,1] := WSTRING#'FINISHED GOODS';   // cv 03
   me.stations[27].raw[44,2] := WSTRING#'16.08.208.041.000A';   // cv 03
   me.stations[27].raw[44,3] := WSTRING#'16.08.208.031.020C';   // cv 03
   me.stations[27].raw[44,4] := WSTRING#'';   // cv 03
   me.stations[27].raw[44,5] := WSTRING#'16.08.211.291.000A';   // cv 03
   me.stations[27].raw[44,6] := WSTRING#'16.08.208.661.000F';   // cv 03
   me.stations[27].raw[44,7] := WSTRING#'16.08.208.651.010B';   // cv 03
   me.stations[27].raw[45,0] := WSTRING#'';   // cv 03
   me.stations[27].raw[45,1] := WSTRING#'FINISHED GOODS';   // cv 03
   me.stations[27].raw[45,2] := WSTRING#'16.18.001.301.010A';   // cv 03
   me.stations[27].raw[45,3] := WSTRING#'16.18.011.301.020B';   // cv 03
   me.stations[27].raw[45,4] := WSTRING#'';   // cv 03
   me.stations[27].raw[45,5] := WSTRING#'16.18.008.301.020A';   // cv 03
   me.stations[27].raw[45,6] := WSTRING#'16.18.008.301.030A';   // cv 03
   me.stations[27].raw[45,7] := WSTRING#'16.18.012.401.020A';   // cv 03
   me.stations[27].raw[46,0] := WSTRING#'';   // cv 03
   me.stations[27].raw[46,1] := WSTRING#'FINISHED GOODS';   // cv 03
   me.stations[27].raw[46,2] := WSTRING#'';   // cv 03
   me.stations[27].raw[46,3] := WSTRING#'';   // cv 03
   me.stations[27].raw[46,4] := WSTRING#'';   // cv 03
   me.stations[27].raw[46,5] := WSTRING#'';   // cv 03
   me.stations[27].raw[46,6] := WSTRING#'';   // cv 03
   me.stations[27].raw[46,7] := WSTRING#'';   // cv 03
   me.stations[27].raw[47,0] := WSTRING#'';   // cv 03
   me.stations[27].raw[47,1] := WSTRING#'FINISHED GOODS';   // cv 03
   me.stations[27].raw[47,2] := WSTRING#'';   // cv 03
   me.stations[27].raw[47,3] := WSTRING#'';   // cv 03
   me.stations[27].raw[47,4] := WSTRING#'';   // cv 03
   me.stations[27].raw[47,5] := WSTRING#'';   // cv 03
   me.stations[27].raw[47,6] := WSTRING#'';   // cv 03
   me.stations[27].raw[47,7] := WSTRING#'';   // cv 03
   me.stations[27].raw[48,0] := WSTRING#'';   // cv 03
   me.stations[27].raw[48,1] := WSTRING#'FINISHED GOODS';   // cv 03
   me.stations[27].raw[48,2] := WSTRING#'';   // cv 03
   me.stations[27].raw[48,3] := WSTRING#'';   // cv 03
   me.stations[27].raw[48,4] := WSTRING#'';   // cv 03
   me.stations[27].raw[48,5] := WSTRING#'';   // cv 03
   me.stations[27].raw[48,6] := WSTRING#'';   // cv 03
   me.stations[27].raw[48,7] := WSTRING#'';   // cv 03
   me.stations[27].raw[49,0] := WSTRING#'';   // cv 03
   me.stations[27].raw[49,1] := WSTRING#'FINISHED GOODS';   // cv 03
   me.stations[27].raw[49,2] := WSTRING#'';   // cv 03
   me.stations[27].raw[49,3] := WSTRING#'';   // cv 03
   me.stations[27].raw[49,4] := WSTRING#'';   // cv 03
   me.stations[27].raw[49,5] := WSTRING#'';   // cv 03
   me.stations[27].raw[49,6] := WSTRING#'';   // cv 03
   me.stations[27].raw[49,7] := WSTRING#'';   // cv 03
   me.stations[28].size := 11;   // cv 04
   me.stations[28].wip[8] := WSTRING#'16.08.208.651.000G$LStuffed Shell SCR- NGK';   // cv 04
   me.stations[28].wip[9] := WSTRING#'16.08.211.806.400B$LSA DPF Stuffed Shell';   // cv 04
   me.stations[28].wip[10] := WSTRING#'16.08.216.806.400A$L DPF Sleeved 2016';   // cv 04
   me.stations[28].wip[11] := WSTRING#'';   // cv 04
   me.stations[28].wip[12] := WSTRING#'';   // cv 04
   me.stations[28].wip[13] := WSTRING#'';   // cv 04
   me.stations[28].wip[14] := WSTRING#'';   // cv 04
   me.stations[28].wip[15] := WSTRING#'';   // cv 04
   me.stations[28].wip[16] := WSTRING#'';   // cv 04
   me.stations[28].wip[17] := WSTRING#'';   // cv 04
   me.stations[28].wip[18] := WSTRING#'';   // cv 04
   me.stations[28].wip[19] := WSTRING#'';   // cv 04
   me.stations[28].wip[20] := WSTRING#'';   // cv 04
   me.stations[28].wip[21] := WSTRING#'';   // cv 04
   me.stations[28].wip[22] := WSTRING#'';   // cv 04
   me.stations[28].wip[23] := WSTRING#'';   // cv 04
   me.stations[28].wip[24] := WSTRING#'';   // cv 04
   me.stations[28].wip[25] := WSTRING#'';   // cv 04
   me.stations[28].wip[26] := WSTRING#'';   // cv 04
   me.stations[28].wip[27] := WSTRING#'';   // cv 04
   me.stations[28].wip[28] := WSTRING#'';   // cv 04
   me.stations[28].wip[29] := WSTRING#'';   // cv 04
   me.stations[28].wip[30] := WSTRING#'';   // cv 04
   me.stations[28].wip[31] := WSTRING#'';   // cv 04
   me.stations[28].wip[32] := WSTRING#'';   // cv 04
   me.stations[28].wip[33] := WSTRING#'';   // cv 04
   me.stations[28].wip[34] := WSTRING#'';   // cv 04
   me.stations[28].wip[35] := WSTRING#'';   // cv 04
   me.stations[28].wip[36] := WSTRING#'';   // cv 04
   me.stations[28].wip[37] := WSTRING#'';   // cv 04
   me.stations[28].wip[38] := WSTRING#'';   // cv 04
   me.stations[28].wip[39] := WSTRING#'';   // cv 04
   me.stations[28].wip[40] := WSTRING#'';   // cv 04
   me.stations[28].wip[41] := WSTRING#'';   // cv 04
   me.stations[28].wip[42] := WSTRING#'';   // cv 04
   me.stations[28].wip[43] := WSTRING#'';   // cv 04
   me.stations[28].wip[44] := WSTRING#'';   // cv 04
   me.stations[28].wip[45] := WSTRING#'';   // cv 04
   me.stations[28].wip[46] := WSTRING#'';   // cv 04
   me.stations[28].wip[47] := WSTRING#'';   // cv 04
   me.stations[28].wip[48] := WSTRING#'';   // cv 04
   me.stations[28].wip[49] := WSTRING#'';   // cv 04
   me.stations[28].raw[8,0] := WSTRING#'';   // cv 04
   me.stations[28].raw[8,1] := WSTRING#'C/O MATERIALS';   // cv 04
   me.stations[28].raw[8,2] := WSTRING#'16.08.208.041.000A';   // cv 04
   me.stations[28].raw[8,3] := WSTRING#'16.08.208.031.020C';   // cv 04
   me.stations[28].raw[8,4] := WSTRING#'';   // cv 04
   me.stations[28].raw[8,5] := WSTRING#'16.08.211.291.000A';   // cv 04
   me.stations[28].raw[8,6] := WSTRING#'16.08.208.661.000F';   // cv 04
   me.stations[28].raw[8,7] := WSTRING#'16.08.208.651.010B';   // cv 04
   me.stations[28].raw[9,0] := WSTRING#'';   // cv 04
   me.stations[28].raw[9,1] := WSTRING#'C/O MATERIALS';   // cv 04
   me.stations[28].raw[9,2] := WSTRING#'16.08.211.806.020A';   // cv 04
   me.stations[28].raw[9,3] := WSTRING#'';   // cv 04
   me.stations[28].raw[9,4] := WSTRING#'';   // cv 04
   me.stations[28].raw[9,5] := WSTRING#'';   // cv 04
   me.stations[28].raw[9,6] := WSTRING#'16.08.208.631.000F';   // cv 04
   me.stations[28].raw[9,7] := WSTRING#'16.08.216.315.000A';   // cv 04
   me.stations[28].raw[10,0] := WSTRING#'';   // cv 04
   me.stations[28].raw[10,1] := WSTRING#'C/O MATERIALS';   // cv 04
   me.stations[28].raw[10,2] := WSTRING#'16.08.216.806.020A';   // cv 04
   me.stations[28].raw[10,3] := WSTRING#'';   // cv 04
   me.stations[28].raw[10,4] := WSTRING#'';   // cv 04
   me.stations[28].raw[10,5] := WSTRING#'';   // cv 04
   me.stations[28].raw[10,6] := WSTRING#'16.08.208.631.000F';   // cv 04
   me.stations[28].raw[10,7] := WSTRING#'16.08.216.315.000A';   // cv 04
   me.stations[28].raw[11,0] := WSTRING#'';   // cv 04
   me.stations[28].raw[11,1] := WSTRING#'';   // cv 04
   me.stations[28].raw[11,2] := WSTRING#'';   // cv 04
   me.stations[28].raw[11,3] := WSTRING#'';   // cv 04
   me.stations[28].raw[11,4] := WSTRING#'';   // cv 04
   me.stations[28].raw[11,5] := WSTRING#'';   // cv 04
   me.stations[28].raw[11,6] := WSTRING#'';   // cv 04
   me.stations[28].raw[11,7] := WSTRING#'';   // cv 04
   me.stations[28].raw[12,0] := WSTRING#'';   // cv 04
   me.stations[28].raw[12,1] := WSTRING#'';   // cv 04
   me.stations[28].raw[12,2] := WSTRING#'';   // cv 04
   me.stations[28].raw[12,3] := WSTRING#'';   // cv 04
   me.stations[28].raw[12,4] := WSTRING#'';   // cv 04
   me.stations[28].raw[12,5] := WSTRING#'';   // cv 04
   me.stations[28].raw[12,6] := WSTRING#'';   // cv 04
   me.stations[28].raw[12,7] := WSTRING#'';   // cv 04
   me.stations[28].raw[13,0] := WSTRING#'';   // cv 04
   me.stations[28].raw[13,1] := WSTRING#'';   // cv 04
   me.stations[28].raw[13,2] := WSTRING#'';   // cv 04
   me.stations[28].raw[13,3] := WSTRING#'';   // cv 04
   me.stations[28].raw[13,4] := WSTRING#'';   // cv 04
   me.stations[28].raw[13,5] := WSTRING#'';   // cv 04
   me.stations[28].raw[13,6] := WSTRING#'';   // cv 04
   me.stations[28].raw[13,7] := WSTRING#'';   // cv 04
   me.stations[28].raw[14,0] := WSTRING#'';   // cv 04
   me.stations[28].raw[14,1] := WSTRING#'';   // cv 04
   me.stations[28].raw[14,2] := WSTRING#'';   // cv 04
   me.stations[28].raw[14,3] := WSTRING#'';   // cv 04
   me.stations[28].raw[14,4] := WSTRING#'';   // cv 04
   me.stations[28].raw[14,5] := WSTRING#'';   // cv 04
   me.stations[28].raw[14,6] := WSTRING#'';   // cv 04
   me.stations[28].raw[14,7] := WSTRING#'';   // cv 04
   me.stations[28].raw[15,0] := WSTRING#'';   // cv 04
   me.stations[28].raw[15,1] := WSTRING#'';   // cv 04
   me.stations[28].raw[15,2] := WSTRING#'';   // cv 04
   me.stations[28].raw[15,3] := WSTRING#'';   // cv 04
   me.stations[28].raw[15,4] := WSTRING#'';   // cv 04
   me.stations[28].raw[15,5] := WSTRING#'';   // cv 04
   me.stations[28].raw[15,6] := WSTRING#'';   // cv 04
   me.stations[28].raw[15,7] := WSTRING#'';   // cv 04
   me.stations[28].raw[16,0] := WSTRING#'';   // cv 04
   me.stations[28].raw[16,1] := WSTRING#'';   // cv 04
   me.stations[28].raw[16,2] := WSTRING#'';   // cv 04
   me.stations[28].raw[16,3] := WSTRING#'';   // cv 04
   me.stations[28].raw[16,4] := WSTRING#'';   // cv 04
   me.stations[28].raw[16,5] := WSTRING#'';   // cv 04
   me.stations[28].raw[16,6] := WSTRING#'';   // cv 04
   me.stations[28].raw[16,7] := WSTRING#'';   // cv 04
   me.stations[28].raw[17,0] := WSTRING#'';   // cv 04
   me.stations[28].raw[17,1] := WSTRING#'';   // cv 04
   me.stations[28].raw[17,2] := WSTRING#'';   // cv 04
   me.stations[28].raw[17,3] := WSTRING#'';   // cv 04
   me.stations[28].raw[17,4] := WSTRING#'';   // cv 04
   me.stations[28].raw[17,5] := WSTRING#'';   // cv 04
   me.stations[28].raw[17,6] := WSTRING#'';   // cv 04
   me.stations[28].raw[17,7] := WSTRING#'';   // cv 04
   me.stations[28].raw[18,0] := WSTRING#'';   // cv 04
   me.stations[28].raw[18,1] := WSTRING#'';   // cv 04
   me.stations[28].raw[18,2] := WSTRING#'';   // cv 04
   me.stations[28].raw[18,3] := WSTRING#'';   // cv 04
   me.stations[28].raw[18,4] := WSTRING#'';   // cv 04
   me.stations[28].raw[18,5] := WSTRING#'';   // cv 04
   me.stations[28].raw[18,6] := WSTRING#'';   // cv 04
   me.stations[28].raw[18,7] := WSTRING#'';   // cv 04
   me.stations[28].raw[19,0] := WSTRING#'';   // cv 04
   me.stations[28].raw[19,1] := WSTRING#'';   // cv 04
   me.stations[28].raw[19,2] := WSTRING#'';   // cv 04
   me.stations[28].raw[19,3] := WSTRING#'';   // cv 04
   me.stations[28].raw[19,4] := WSTRING#'';   // cv 04
   me.stations[28].raw[19,5] := WSTRING#'';   // cv 04
   me.stations[28].raw[19,6] := WSTRING#'';   // cv 04
   me.stations[28].raw[19,7] := WSTRING#'';   // cv 04
   me.stations[28].raw[20,0] := WSTRING#'';   // cv 04
   me.stations[28].raw[20,1] := WSTRING#'';   // cv 04
   me.stations[28].raw[20,2] := WSTRING#'';   // cv 04
   me.stations[28].raw[20,3] := WSTRING#'';   // cv 04
   me.stations[28].raw[20,4] := WSTRING#'';   // cv 04
   me.stations[28].raw[20,5] := WSTRING#'';   // cv 04
   me.stations[28].raw[20,6] := WSTRING#'';   // cv 04
   me.stations[28].raw[20,7] := WSTRING#'';   // cv 04
   me.stations[28].raw[21,0] := WSTRING#'';   // cv 04
   me.stations[28].raw[21,1] := WSTRING#'';   // cv 04
   me.stations[28].raw[21,2] := WSTRING#'';   // cv 04
   me.stations[28].raw[21,3] := WSTRING#'';   // cv 04
   me.stations[28].raw[21,4] := WSTRING#'';   // cv 04
   me.stations[28].raw[21,5] := WSTRING#'';   // cv 04
   me.stations[28].raw[21,6] := WSTRING#'';   // cv 04
   me.stations[28].raw[21,7] := WSTRING#'';   // cv 04
   me.stations[28].raw[22,0] := WSTRING#'';   // cv 04
   me.stations[28].raw[22,1] := WSTRING#'';   // cv 04
   me.stations[28].raw[22,2] := WSTRING#'';   // cv 04
   me.stations[28].raw[22,3] := WSTRING#'';   // cv 04
   me.stations[28].raw[22,4] := WSTRING#'';   // cv 04
   me.stations[28].raw[22,5] := WSTRING#'';   // cv 04
   me.stations[28].raw[22,6] := WSTRING#'';   // cv 04
   me.stations[28].raw[22,7] := WSTRING#'';   // cv 04
   me.stations[28].raw[23,0] := WSTRING#'';   // cv 04
   me.stations[28].raw[23,1] := WSTRING#'';   // cv 04
   me.stations[28].raw[23,2] := WSTRING#'';   // cv 04
   me.stations[28].raw[23,3] := WSTRING#'';   // cv 04
   me.stations[28].raw[23,4] := WSTRING#'';   // cv 04
   me.stations[28].raw[23,5] := WSTRING#'';   // cv 04
   me.stations[28].raw[23,6] := WSTRING#'';   // cv 04
   me.stations[28].raw[23,7] := WSTRING#'';   // cv 04
   me.stations[28].raw[24,0] := WSTRING#'';   // cv 04
   me.stations[28].raw[24,1] := WSTRING#'';   // cv 04
   me.stations[28].raw[24,2] := WSTRING#'';   // cv 04
   me.stations[28].raw[24,3] := WSTRING#'';   // cv 04
   me.stations[28].raw[24,4] := WSTRING#'';   // cv 04
   me.stations[28].raw[24,5] := WSTRING#'';   // cv 04
   me.stations[28].raw[24,6] := WSTRING#'';   // cv 04
   me.stations[28].raw[24,7] := WSTRING#'';   // cv 04
   me.stations[28].raw[25,0] := WSTRING#'';   // cv 04
   me.stations[28].raw[25,1] := WSTRING#'';   // cv 04
   me.stations[28].raw[25,2] := WSTRING#'';   // cv 04
   me.stations[28].raw[25,3] := WSTRING#'';   // cv 04
   me.stations[28].raw[25,4] := WSTRING#'';   // cv 04
   me.stations[28].raw[25,5] := WSTRING#'';   // cv 04
   me.stations[28].raw[25,6] := WSTRING#'';   // cv 04
   me.stations[28].raw[25,7] := WSTRING#'';   // cv 04
   me.stations[28].raw[26,0] := WSTRING#'';   // cv 04
   me.stations[28].raw[26,1] := WSTRING#'';   // cv 04
   me.stations[28].raw[26,2] := WSTRING#'';   // cv 04
   me.stations[28].raw[26,3] := WSTRING#'';   // cv 04
   me.stations[28].raw[26,4] := WSTRING#'';   // cv 04
   me.stations[28].raw[26,5] := WSTRING#'';   // cv 04
   me.stations[28].raw[26,6] := WSTRING#'';   // cv 04
   me.stations[28].raw[26,7] := WSTRING#'';   // cv 04
   me.stations[28].raw[27,0] := WSTRING#'';   // cv 04
   me.stations[28].raw[27,1] := WSTRING#'';   // cv 04
   me.stations[28].raw[27,2] := WSTRING#'';   // cv 04
   me.stations[28].raw[27,3] := WSTRING#'';   // cv 04
   me.stations[28].raw[27,4] := WSTRING#'';   // cv 04
   me.stations[28].raw[27,5] := WSTRING#'';   // cv 04
   me.stations[28].raw[27,6] := WSTRING#'';   // cv 04
   me.stations[28].raw[27,7] := WSTRING#'';   // cv 04
   me.stations[28].raw[28,0] := WSTRING#'';   // cv 04
   me.stations[28].raw[28,1] := WSTRING#'';   // cv 04
   me.stations[28].raw[28,2] := WSTRING#'';   // cv 04
   me.stations[28].raw[28,3] := WSTRING#'';   // cv 04
   me.stations[28].raw[28,4] := WSTRING#'';   // cv 04
   me.stations[28].raw[28,5] := WSTRING#'';   // cv 04
   me.stations[28].raw[28,6] := WSTRING#'';   // cv 04
   me.stations[28].raw[28,7] := WSTRING#'';   // cv 04
   me.stations[28].raw[29,0] := WSTRING#'';   // cv 04
   me.stations[28].raw[29,1] := WSTRING#'';   // cv 04
   me.stations[28].raw[29,2] := WSTRING#'';   // cv 04
   me.stations[28].raw[29,3] := WSTRING#'';   // cv 04
   me.stations[28].raw[29,4] := WSTRING#'';   // cv 04
   me.stations[28].raw[29,5] := WSTRING#'';   // cv 04
   me.stations[28].raw[29,6] := WSTRING#'';   // cv 04
   me.stations[28].raw[29,7] := WSTRING#'';   // cv 04
   me.stations[28].raw[30,0] := WSTRING#'';   // cv 04
   me.stations[28].raw[30,1] := WSTRING#'';   // cv 04
   me.stations[28].raw[30,2] := WSTRING#'';   // cv 04
   me.stations[28].raw[30,3] := WSTRING#'';   // cv 04
   me.stations[28].raw[30,4] := WSTRING#'';   // cv 04
   me.stations[28].raw[30,5] := WSTRING#'';   // cv 04
   me.stations[28].raw[30,6] := WSTRING#'';   // cv 04
   me.stations[28].raw[30,7] := WSTRING#'';   // cv 04
   me.stations[28].raw[31,0] := WSTRING#'';   // cv 04
   me.stations[28].raw[31,1] := WSTRING#'';   // cv 04
   me.stations[28].raw[31,2] := WSTRING#'';   // cv 04
   me.stations[28].raw[31,3] := WSTRING#'';   // cv 04
   me.stations[28].raw[31,4] := WSTRING#'';   // cv 04
   me.stations[28].raw[31,5] := WSTRING#'';   // cv 04
   me.stations[28].raw[31,6] := WSTRING#'';   // cv 04
   me.stations[28].raw[31,7] := WSTRING#'';   // cv 04
   me.stations[28].raw[32,0] := WSTRING#'';   // cv 04
   me.stations[28].raw[32,1] := WSTRING#'';   // cv 04
   me.stations[28].raw[32,2] := WSTRING#'';   // cv 04
   me.stations[28].raw[32,3] := WSTRING#'';   // cv 04
   me.stations[28].raw[32,4] := WSTRING#'';   // cv 04
   me.stations[28].raw[32,5] := WSTRING#'';   // cv 04
   me.stations[28].raw[32,6] := WSTRING#'';   // cv 04
   me.stations[28].raw[32,7] := WSTRING#'';   // cv 04
   me.stations[28].raw[33,0] := WSTRING#'';   // cv 04
   me.stations[28].raw[33,1] := WSTRING#'';   // cv 04
   me.stations[28].raw[33,2] := WSTRING#'';   // cv 04
   me.stations[28].raw[33,3] := WSTRING#'';   // cv 04
   me.stations[28].raw[33,4] := WSTRING#'';   // cv 04
   me.stations[28].raw[33,5] := WSTRING#'';   // cv 04
   me.stations[28].raw[33,6] := WSTRING#'';   // cv 04
   me.stations[28].raw[33,7] := WSTRING#'';   // cv 04
   me.stations[28].raw[34,0] := WSTRING#'';   // cv 04
   me.stations[28].raw[34,1] := WSTRING#'';   // cv 04
   me.stations[28].raw[34,2] := WSTRING#'';   // cv 04
   me.stations[28].raw[34,3] := WSTRING#'';   // cv 04
   me.stations[28].raw[34,4] := WSTRING#'';   // cv 04
   me.stations[28].raw[34,5] := WSTRING#'';   // cv 04
   me.stations[28].raw[34,6] := WSTRING#'';   // cv 04
   me.stations[28].raw[34,7] := WSTRING#'';   // cv 04
   me.stations[28].raw[35,0] := WSTRING#'';   // cv 04
   me.stations[28].raw[35,1] := WSTRING#'';   // cv 04
   me.stations[28].raw[35,2] := WSTRING#'';   // cv 04
   me.stations[28].raw[35,3] := WSTRING#'';   // cv 04
   me.stations[28].raw[35,4] := WSTRING#'';   // cv 04
   me.stations[28].raw[35,5] := WSTRING#'';   // cv 04
   me.stations[28].raw[35,6] := WSTRING#'';   // cv 04
   me.stations[28].raw[35,7] := WSTRING#'';   // cv 04
   me.stations[28].raw[36,0] := WSTRING#'';   // cv 04
   me.stations[28].raw[36,1] := WSTRING#'';   // cv 04
   me.stations[28].raw[36,2] := WSTRING#'';   // cv 04
   me.stations[28].raw[36,3] := WSTRING#'';   // cv 04
   me.stations[28].raw[36,4] := WSTRING#'';   // cv 04
   me.stations[28].raw[36,5] := WSTRING#'';   // cv 04
   me.stations[28].raw[36,6] := WSTRING#'';   // cv 04
   me.stations[28].raw[36,7] := WSTRING#'';   // cv 04
   me.stations[28].raw[37,0] := WSTRING#'';   // cv 04
   me.stations[28].raw[37,1] := WSTRING#'';   // cv 04
   me.stations[28].raw[37,2] := WSTRING#'';   // cv 04
   me.stations[28].raw[37,3] := WSTRING#'';   // cv 04
   me.stations[28].raw[37,4] := WSTRING#'';   // cv 04
   me.stations[28].raw[37,5] := WSTRING#'';   // cv 04
   me.stations[28].raw[37,6] := WSTRING#'';   // cv 04
   me.stations[28].raw[37,7] := WSTRING#'';   // cv 04
   me.stations[28].raw[38,0] := WSTRING#'';   // cv 04
   me.stations[28].raw[38,1] := WSTRING#'';   // cv 04
   me.stations[28].raw[38,2] := WSTRING#'';   // cv 04
   me.stations[28].raw[38,3] := WSTRING#'';   // cv 04
   me.stations[28].raw[38,4] := WSTRING#'';   // cv 04
   me.stations[28].raw[38,5] := WSTRING#'';   // cv 04
   me.stations[28].raw[38,6] := WSTRING#'';   // cv 04
   me.stations[28].raw[38,7] := WSTRING#'';   // cv 04
   me.stations[28].raw[39,0] := WSTRING#'';   // cv 04
   me.stations[28].raw[39,1] := WSTRING#'';   // cv 04
   me.stations[28].raw[39,2] := WSTRING#'';   // cv 04
   me.stations[28].raw[39,3] := WSTRING#'';   // cv 04
   me.stations[28].raw[39,4] := WSTRING#'';   // cv 04
   me.stations[28].raw[39,5] := WSTRING#'';   // cv 04
   me.stations[28].raw[39,6] := WSTRING#'';   // cv 04
   me.stations[28].raw[39,7] := WSTRING#'';   // cv 04
   me.stations[28].raw[40,0] := WSTRING#'';   // cv 04
   me.stations[28].raw[40,1] := WSTRING#'';   // cv 04
   me.stations[28].raw[40,2] := WSTRING#'';   // cv 04
   me.stations[28].raw[40,3] := WSTRING#'';   // cv 04
   me.stations[28].raw[40,4] := WSTRING#'';   // cv 04
   me.stations[28].raw[40,5] := WSTRING#'';   // cv 04
   me.stations[28].raw[40,6] := WSTRING#'';   // cv 04
   me.stations[28].raw[40,7] := WSTRING#'';   // cv 04
   me.stations[28].raw[41,0] := WSTRING#'';   // cv 04
   me.stations[28].raw[41,1] := WSTRING#'';   // cv 04
   me.stations[28].raw[41,2] := WSTRING#'';   // cv 04
   me.stations[28].raw[41,3] := WSTRING#'';   // cv 04
   me.stations[28].raw[41,4] := WSTRING#'';   // cv 04
   me.stations[28].raw[41,5] := WSTRING#'';   // cv 04
   me.stations[28].raw[41,6] := WSTRING#'';   // cv 04
   me.stations[28].raw[41,7] := WSTRING#'';   // cv 04
   me.stations[28].raw[42,0] := WSTRING#'';   // cv 04
   me.stations[28].raw[42,1] := WSTRING#'';   // cv 04
   me.stations[28].raw[42,2] := WSTRING#'';   // cv 04
   me.stations[28].raw[42,3] := WSTRING#'';   // cv 04
   me.stations[28].raw[42,4] := WSTRING#'';   // cv 04
   me.stations[28].raw[42,5] := WSTRING#'';   // cv 04
   me.stations[28].raw[42,6] := WSTRING#'';   // cv 04
   me.stations[28].raw[42,7] := WSTRING#'';   // cv 04
   me.stations[28].raw[43,0] := WSTRING#'';   // cv 04
   me.stations[28].raw[43,1] := WSTRING#'';   // cv 04
   me.stations[28].raw[43,2] := WSTRING#'';   // cv 04
   me.stations[28].raw[43,3] := WSTRING#'';   // cv 04
   me.stations[28].raw[43,4] := WSTRING#'';   // cv 04
   me.stations[28].raw[43,5] := WSTRING#'';   // cv 04
   me.stations[28].raw[43,6] := WSTRING#'';   // cv 04
   me.stations[28].raw[43,7] := WSTRING#'';   // cv 04
   me.stations[28].raw[44,0] := WSTRING#'';   // cv 04
   me.stations[28].raw[44,1] := WSTRING#'';   // cv 04
   me.stations[28].raw[44,2] := WSTRING#'';   // cv 04
   me.stations[28].raw[44,3] := WSTRING#'';   // cv 04
   me.stations[28].raw[44,4] := WSTRING#'';   // cv 04
   me.stations[28].raw[44,5] := WSTRING#'';   // cv 04
   me.stations[28].raw[44,6] := WSTRING#'';   // cv 04
   me.stations[28].raw[44,7] := WSTRING#'';   // cv 04
   me.stations[28].raw[45,0] := WSTRING#'';   // cv 04
   me.stations[28].raw[45,1] := WSTRING#'';   // cv 04
   me.stations[28].raw[45,2] := WSTRING#'';   // cv 04
   me.stations[28].raw[45,3] := WSTRING#'';   // cv 04
   me.stations[28].raw[45,4] := WSTRING#'';   // cv 04
   me.stations[28].raw[45,5] := WSTRING#'';   // cv 04
   me.stations[28].raw[45,6] := WSTRING#'';   // cv 04
   me.stations[28].raw[45,7] := WSTRING#'';   // cv 04
   me.stations[28].raw[46,0] := WSTRING#'';   // cv 04
   me.stations[28].raw[46,1] := WSTRING#'';   // cv 04
   me.stations[28].raw[46,2] := WSTRING#'';   // cv 04
   me.stations[28].raw[46,3] := WSTRING#'';   // cv 04
   me.stations[28].raw[46,4] := WSTRING#'';   // cv 04
   me.stations[28].raw[46,5] := WSTRING#'';   // cv 04
   me.stations[28].raw[46,6] := WSTRING#'';   // cv 04
   me.stations[28].raw[46,7] := WSTRING#'';   // cv 04
   me.stations[28].raw[47,0] := WSTRING#'';   // cv 04
   me.stations[28].raw[47,1] := WSTRING#'';   // cv 04
   me.stations[28].raw[47,2] := WSTRING#'';   // cv 04
   me.stations[28].raw[47,3] := WSTRING#'';   // cv 04
   me.stations[28].raw[47,4] := WSTRING#'';   // cv 04
   me.stations[28].raw[47,5] := WSTRING#'';   // cv 04
   me.stations[28].raw[47,6] := WSTRING#'';   // cv 04
   me.stations[28].raw[47,7] := WSTRING#'';   // cv 04
   me.stations[28].raw[48,0] := WSTRING#'';   // cv 04
   me.stations[28].raw[48,1] := WSTRING#'';   // cv 04
   me.stations[28].raw[48,2] := WSTRING#'';   // cv 04
   me.stations[28].raw[48,3] := WSTRING#'';   // cv 04
   me.stations[28].raw[48,4] := WSTRING#'';   // cv 04
   me.stations[28].raw[48,5] := WSTRING#'';   // cv 04
   me.stations[28].raw[48,6] := WSTRING#'';   // cv 04
   me.stations[28].raw[48,7] := WSTRING#'';   // cv 04
   me.stations[28].raw[49,0] := WSTRING#'';   // cv 04
   me.stations[28].raw[49,1] := WSTRING#'';   // cv 04
   me.stations[28].raw[49,2] := WSTRING#'';   // cv 04
   me.stations[28].raw[49,3] := WSTRING#'';   // cv 04
   me.stations[28].raw[49,4] := WSTRING#'';   // cv 04
   me.stations[28].raw[49,5] := WSTRING#'';   // cv 04
   me.stations[28].raw[49,6] := WSTRING#'';   // cv 04
   me.stations[28].raw[49,7] := WSTRING#'';   // cv 04
   me.stations[29].size := 3;
   me.stations[29].wip[3] := WSTRING#'';
   me.stations[29].wip[4] := WSTRING#'';
   me.stations[29].wip[5] := WSTRING#'';
   me.stations[29].wip[6] := WSTRING#'';
   me.stations[29].wip[7] := WSTRING#'';
   me.stations[29].wip[8] := WSTRING#'';
   me.stations[29].wip[9] := WSTRING#'';
   me.stations[29].wip[10] := WSTRING#'';
   me.stations[29].wip[11] := WSTRING#'';
   me.stations[29].wip[12] := WSTRING#'';
   me.stations[29].wip[13] := WSTRING#'';
   me.stations[29].wip[14] := WSTRING#'';
   me.stations[29].wip[15] := WSTRING#'';
   me.stations[29].wip[16] := WSTRING#'';
   me.stations[29].wip[17] := WSTRING#'';
   me.stations[29].wip[18] := WSTRING#'';
   me.stations[29].wip[19] := WSTRING#'';
   me.stations[29].wip[20] := WSTRING#'';
   me.stations[29].wip[21] := WSTRING#'';
   me.stations[29].wip[22] := WSTRING#'';
